# B&R Automation Studio project NAEUL004C00R13L518F00 (part 26)

#### Act_OptP1026Lifter2FBCtrl.st
```iecst
ACTION Act_OptP1026Lifter2FBCtrl:

	fbJogSlowToFastDlyTm.PT	:= T#2s;
	fbJogSlowToFastDlyTm;
	fbLmtRstTm;

	//Lifter Safety Sensor Interruption
	IF EDGENEG(p_tyDI.bLifterSafetyLmtSW1 AND p_tyDI.bLifterSafetyLmtSW2 AND p_tyDI.bLifterTimingBeltSen) THEN
		tyP1026McSetTeach.tyMotionStdLifter.tyBtnStop.bRtCompl	:= TRUE;
	END_IF

	IF EDGEPOS((p_udiLifter2AxisErrID = 21570 OR p_udiLifter2AxisErrID = 21571) AND tyP1026McSetTeach.tyMotionStdLifter.tyBtnJogDown.bValue = FALSE AND tyP1026McSetTeach.tyMotionStdLifter.tyBtnJogUp.bValue = FALSE) THEN
		fbLmtRstTm.IN	:= TRUE;
	END_IF

	IF fbLmtRstTm.Q = TRUE THEN
		tyP1026McSetTeach.tyMotionStdLifter.tyBtnRst.bRtCompl	:= TRUE;
	END_IF

	IF (tyP1026McSetTeach.tyMotionStdLifter.tyBtnJogUp.bValue = FALSE AND tyP1026McSetTeach.tyMotionStdLifter.tyBtnJogDown.bValue = FALSE) AND (p_bLifter2Jogging = TRUE) THEN
		bJogStopLifter	:= TRUE;
	END_IF

	IF tyP1026McSetTeach.tyMotionStdLifter.tyBtnStop.bRtCompl = TRUE THEN
		eLifter2Act		:= LifterActStop;

		IF p_eLifter2Stat = LifterActStop AND p_eLifter2Status = Done THEN
			eLifter2Act	:= LifterActIdle;

			tyP1026McSetTeach.tyMotionStdLifter.tyBtnStop.bRtCompl			:= FALSE;
			tyP1026McSetTeach.tyMotionStdLifter.tyBtnJogDown.bRtCompl		:= FALSE;
			tyP1026McSetTeach.tyMotionStdLifter.tyBtnJogUp.bRtCompl			:= FALSE;
			tyP1026McSetTeach.tyMotionStdLifter.tyBtnOrigin.bRtCompl		:= FALSE;
			tyP1026McSetTeach.tyMotionStdLifter.tyBtnMovAbs.bRtCompl		:= FALSE;
			tyP1026McSetTeach.tyMotionStdLifter.tyBtnMovRel.bRtCompl		:= FALSE;

			tyP1026McSetTeach.tyTeachLifterTopPos2.tyBtn2.bRtCompl				:= FALSE;//
			tyP1026McSetTeach.tyTeachLifterBtmPos2.tyBtn2.bRtCompl				:= FALSE;//

			tyP1026McSetTeach.tyMotionStdLifter.tyBtnStop.bValue			:= TRUE;
			tyP1026McSetTeach.tyMotionStdLifter.tyBtnJogDown.bValue			:= FALSE;
			tyP1026McSetTeach.tyMotionStdLifter.tyBtnJogUp.bValue			:= FALSE;
			tyP1026McSetTeach.tyMotionStdLifter.tyBtnOrigin.bValue			:= FALSE;
			tyP1026McSetTeach.tyMotionStdLifter.tyBtnMovAbs.bValue			:= FALSE;
			tyP1026McSetTeach.tyMotionStdLifter.tyBtnMovRel.bValue			:= FALSE;

			tyP1026McSetTeach.tyTeachLifterTopPos2.tyBtn2.bValue				:= FALSE;
			tyP1026McSetTeach.tyTeachLifterBtmPos2.tyBtn2.bValue				:= FALSE;

			tyP1026McSetTeach.tyMotionStdLifter.tyBtnStop.bRtLk				:= TRUE;
			tyP1026McSetTeach.tyMotionStdLifter.tyBtnJogDown.bRtLk			:= FALSE;
			tyP1026McSetTeach.tyMotionStdLifter.tyBtnJogUp.bRtLk			:= FALSE;
			tyP1026McSetTeach.tyMotionStdLifter.tyBtnOrigin.bRtLk			:= FALSE;
			tyP1026McSetTeach.tyMotionStdLifter.tyBtnMovAbs.bRtLk			:= FALSE;
			tyP1026McSetTeach.tyMotionStdLifter.tyBtnMovRel.bRtLk			:= FALSE;

			tyP1026McSetTeach.tyTeachLifterTopPos2.tyBtn2.bRtLk				:= FALSE;
			tyP1026McSetTeach.tyTeachLifterBtmPos2.tyBtn2.bRtLk				:= FALSE;

		END_IF

	ELSIF (tyP1026McSetTeach.tyMotionStdLifter.tyBtnJogDown.bRtCompl = TRUE) OR (tyP1026McSetTeach.tyMotionStdLifter.tyBtnJogUp.bRtCompl = TRUE) OR (bJogStopLifter = TRUE) THEN
		bJogSlow					:= FALSE;
		bJogFast					:= FALSE;
		fbJogSlowToFastDlyTm.IN		:= FALSE;

		eLifter2Act	:= LifterActJogStop;

		IF p_eLifter2Stat = LifterActJogStop AND p_eLifter2Status = Done THEN
			eLifter2Act		:= LifterActIdle;

			bJogStopLifter	:= FALSE;

			tyP1026McSetTeach.tyMotionStdLifter.tyBtnStop.bRtCompl			:= FALSE;
			tyP1026McSetTeach.tyMotionStdLifter.tyBtnJogDown.bRtCompl		:= FALSE;
			tyP1026McSetTeach.tyMotionStdLifter.tyBtnJogUp.bRtCompl			:= FALSE;
			tyP1026McSetTeach.tyMotionStdLifter.tyBtnOrigin.bRtCompl		:= FALSE;
			tyP1026McSetTeach.tyMotionStdLifter.tyBtnMovAbs.bRtCompl		:= FALSE;
			tyP1026McSetTeach.tyMotionStdLifter.tyBtnMovRel.bRtCompl		:= FALSE;

			tyP1026McSetTeach.tyTeachLifterTopPos2.tyBtn2.bRtCompl				:= FALSE;//
			tyP1026McSetTeach.tyTeachLifterBtmPos2.tyBtn2.bRtCompl				:= FALSE;//

			tyP1026McSetTeach.tyMotionStdLifter.tyBtnStop.bValue			:= TRUE;
			tyP1026McSetTeach.tyMotionStdLifter.tyBtnJogDown.bValue			:= FALSE;
			tyP1026McSetTeach.tyMotionStdLifter.tyBtnJogUp.bValue			:= FALSE;
			tyP1026McSetTeach.tyMotionStdLifter.tyBtnOrigin.bValue			:= FALSE;
			tyP1026McSetTeach.tyMotionStdLifter.tyBtnMovAbs.bValue			:= FALSE;
			tyP1026McSetTeach.tyMotionStdLifter.tyBtnMovRel.bValue			:= FALSE;

			tyP1026McSetTeach.tyTeachLifterTopPos2.tyBtn2.bValue				:= FALSE;
			tyP1026McSetTeach.tyTeachLifterBtmPos2.tyBtn2.bValue				:= FALSE;

			tyP1026McSetTeach.tyMotionStdLifter.tyBtnStop.bRtLk				:= TRUE;
			tyP1026McSetTeach.tyMotionStdLifter.tyBtnJogDown.bRtLk			:= FALSE;
			tyP1026McSetTeach.tyMotionStdLifter.tyBtnJogUp.bRtLk			:= FALSE;
			tyP1026McSetTeach.tyMotionStdLifter.tyBtnOrigin.bRtLk			:= FALSE;
			tyP1026McSetTeach.tyMotionStdLifter.tyBtnMovAbs.bRtLk			:= FALSE;
			tyP1026McSetTeach.tyMotionStdLifter.tyBtnMovRel.bRtLk			:= FALSE;

			tyP1026McSetTeach.tyTeachLifterTopPos2.tyBtn2.bRtLk				:= FALSE;
			tyP1026McSetTeach.tyTeachLifterBtmPos2.tyBtn2.bRtLk				:= FALSE;

		END_IF

	ELSIF tyP1026McSetTeach.tyMotionStdLifter.tyBtnPwr.bRtCompl = TRUE THEN
		tyP1026McSetTeach.tyMotionStdLifter.tyBtnPwr.bRtLk	:= TRUE;

		IF tyP1026McSetTeach.tyMotionStdLifter.tyBtnPwr.bValue = TRUE THEN
			eLifter2Act	:= LifterActPwrOn;

			IF p_eLifter2Stat = LifterActPwrOn AND p_eLifter2Status = Done THEN
				eLifter2Act	:= LifterActIdle;

				tyP1026McSetTeach.tyMotionStdLifter.tyBtnPwr.bRtCompl	:= FALSE;
				tyP1026McSetTeach.tyMotionStdLifter.tyBtnPwr.bRtLk		:= FALSE;
			END_IF
		ELSE
			eLifter2Act	:= LifterActPwrOff;

			IF p_eLifter2Stat = LifterActPwrOff AND p_eLifter2Status = Done THEN
				eLifter2Act	:= LifterActIdle;

				tyP1026McSetTeach.tyMotionStdLifter.tyBtnPwr.bRtCompl	:= FALSE;
				tyP1026McSetTeach.tyMotionStdLifter.tyBtnPwr.bRtLk		:= FALSE;
			END_IF
		END_IF

	ELSIF tyP1026McSetTeach.tyMotionStdLifter.tyBtnOrigin.bRtCompl = TRUE THEN
		tyP1026McSetTeach.tyMotionStdLifter.tyBtnOrigin.bValue	:= TRUE;
		tyP1026McSetTeach.tyMotionStdLifter.tyBtnStop.bValue	:= FALSE;

		tyP1026McSetTeach.tyMotionStdLifter.tyBtnOrigin.bRtLk	:= TRUE;
		tyP1026McSetTeach.tyMotionStdLifter.tyBtnStop.bRtLk		:= FALSE;

		eLifter2Act	:= LifterActHoming;

		IF p_eLifter2Stat = LifterActHoming AND p_eLifter2Status = Done THEN
			eLifter2Act	:= LifterActIdle;

			tyP1026McSetTeach.tyMotionStdLifter.tyBtnOrigin.bRtCompl	:= FALSE;
			tyP1026McSetTeach.tyMotionStdLifter.tyBtnOrigin.bValue		:= FALSE;
			tyP1026McSetTeach.tyMotionStdLifter.tyBtnStop.bValue		:= TRUE;

			tyP1026McSetTeach.tyMotionStdLifter.tyBtnOrigin.bRtLk		:= FALSE;
			tyP1026McSetTeach.tyMotionStdLifter.tyBtnStop.bRtLk			:= TRUE;

		END_IF

	ELSIF tyP1026McSetTeach.tyMotionStdLifter.tyBtnRst.bRtCompl = TRUE THEN
		tyP1026McSetTeach.tyMotionStdLifter.tyBtnRst.bValue	:= TRUE;
		tyP1026McSetTeach.tyMotionStdLifter.tyBtnRst.bRtLk	:= TRUE;

		eLifter2Act	:= LifterActRstAxisErr;

		IF p_eLifter2Stat = LifterActRstAxisErr AND p_eLifter2Status = Done THEN
			eLifter2Act	:= LifterActIdle;

			tyP1026McSetTeach.tyMotionStdLifter.tyBtnRst.bRtCompl	:= FALSE;
			tyP1026McSetTeach.tyMotionStdLifter.tyBtnRst.bValue		:= FALSE;
			tyP1026McSetTeach.tyMotionStdLifter.tyBtnRst.bRtLk		:= FALSE;

			fbLmtRstTm.IN	:= FALSE;
		END_IF

	ELSIF tyP1026McSetTeach.tyTeachLifterTopPos2.tyBtn2.bRtCompl = TRUE THEN
		tyP1026McSetTeach.tyTeachLifterTopPos2.tyBtn2.bValue		:= TRUE;
		tyP1026McSetTeach.tyMotionStdLifter.tyBtnStop.bValue	:= FALSE;

		tyP1026McSetTeach.tyTeachLifterTopPos2.tyBtn2.bRtLk		:= TRUE;
		tyP1026McSetTeach.tyMotionStdLifter.tyBtnStop.bRtLk		:= FALSE;

		diMnlLifterNomSpd2	:= tyP1026McSetTeach.tyMotionStdLifter.tyNumNomSpd.diValue;

		eLifter2Act		:= LifterActGoGPos;

		IF p_eLifter2Stat = LifterActGoGPos AND p_eLifter2Status = Done THEN
			eLifter2Act	:= LifterActIdle;

			tyP1026McSetTeach.tyTeachLifterTopPos2.tyBtn2.bRtCompl		:= FALSE;
			tyP1026McSetTeach.tyTeachLifterTopPos2.tyBtn2.bValue		:= FALSE;
			tyP1026McSetTeach.tyMotionStdLifter.tyBtnStop.bValue	:= TRUE;

			tyP1026McSetTeach.tyTeachLifterTopPos2.tyBtn2.bRtLk		:= FALSE;
			tyP1026McSetTeach.tyMotionStdLifter.tyBtnStop.bRtLk		:= TRUE;
		END_IF

	ELSIF tyP1026McSetTeach.tyTeachLifterBtmPos2.tyBtn2.bRtCompl = TRUE THEN
		tyP1026McSetTeach.tyTeachLifterBtmPos2.tyBtn2.bValue		:= TRUE;
		tyP1026McSetTeach.tyMotionStdLifter.tyBtnStop.bValue	:= FALSE;

		tyP1026McSetTeach.tyTeachLifterBtmPos2.tyBtn2.bRtLk		:= TRUE;
		tyP1026McSetTeach.tyMotionStdLifter.tyBtnStop.bRtLk		:= FALSE;

		diMnlLifterNomSpd2	:= tyP1026McSetTeach.tyMotionStdLifter.tyNumNomSpd.diValue;

		eLifter2Act		:= LifterActGoHPos;

		IF p_eLifter2Stat = LifterActGoHPos AND p_eLifter2Status = Done THEN
			eLifter2Act	:= LifterActIdle;

			tyP1026McSetTeach.tyTeachLifterBtmPos2.tyBtn2.bRtCompl		:= FALSE;
			tyP1026McSetTeach.tyTeachLifterBtmPos2.tyBtn2.bValue		:= FALSE;
			tyP1026McSetTeach.tyMotionStdLifter.tyBtnStop.bValue	:= TRUE;

			tyP1026McSetTeach.tyTeachLifterBtmPos2.tyBtn2.bRtLk		:= FALSE;
			tyP1026McSetTeach.tyMotionStdLifter.tyBtnStop.bRtLk		:= TRUE;
		END_IF

	ELSIF tyP1026McSetTeach.tyMotionStdLifter.tyBtnMovAbs.bRtCompl = TRUE THEN

		tyP1026McSetTeach.tyMotionStdLifter.tyBtnMovAbs.bValue	:= TRUE;
		tyP1026McSetTeach.tyMotionStdLifter.tyBtnStop.bValue	:= FALSE;

		tyP1026McSetTeach.tyMotionStdLifter.tyBtnMovAbs.bRtLk	:= TRUE;
		tyP1026McSetTeach.tyMotionStdLifter.tyBtnStop.bRtLk		:= FALSE;

		diMnlLifterTargetPos2	:= tyP1026McSetTeach.tyMotionStdLifter.tyNumTargetPos.diValue;
		diMnlLifterNomSpd2		:= tyP1026McSetTeach.tyMotionStdLifter.tyNumNomSpd.diValue;

		eLifter2Act			:= LifterActMovAbs;

		IF p_eLifter2Stat = LifterActMovAbs AND p_eLifter2Status = Done THEN
			eLifter2Act	:= LifterActIdle;

			tyP1026McSetTeach.tyMotionStdLifter.tyBtnMovAbs.bRtCompl	:= FALSE;
			tyP1026McSetTeach.tyMotionStdLifter.tyBtnMovAbs.bValue		:= FALSE;
			tyP1026McSetTeach.tyMotionStdLifter.tyBtnStop.bValue		:= TRUE;

			tyP1026McSetTeach.tyMotionStdLifter.tyBtnMovAbs.bRtLk		:= FALSE;
			tyP1026McSetTeach.tyMotionStdLifter.tyBtnStop.bRtLk			:= TRUE;
		END_IF

	ELSIF tyP1026McSetTeach.tyMotionStdLifter.tyBtnMovRel.bRtCompl = TRUE THEN
		tyP1026McSetTeach.tyMotionStdLifter.tyBtnMovRel.bValue			:= TRUE;
		tyP1026McSetTeach.tyMotionStdLifter.tyBtnStop.bValue			:= FALSE;

		tyP1026McSetTeach.tyMotionStdLifter.tyBtnMovRel.bRtLk			:= TRUE;
		tyP1026McSetTeach.tyMotionStdLifter.tyBtnStop.bRtLk				:= FALSE;

		diMnlLifterStepSize2		:= tyP1026McSetTeach.tyMotionStdLifter.tyNumStepSize.diValue;
		diMnlLifterNomSpd2		:= tyP1026McSetTeach.tyMotionStdLifter.tyNumNomSpd.diValue;

		eLifter2Act		:= LifterActMovRel;

		IF p_eLifter2Stat = LifterActMovRel AND p_eLifter2Status = Done THEN
			eLifter2Act	:= LifterActIdle;

			tyP1026McSetTeach.tyMotionStdLifter.tyBtnMovRel.bRtCompl		:= FALSE;
			tyP1026McSetTeach.tyMotionStdLifter.tyBtnMovRel.bValue			:= FALSE;
			tyP1026McSetTeach.tyMotionStdLifter.tyBtnStop.bValue			:= TRUE;

			tyP1026McSetTeach.tyMotionStdLifter.tyBtnMovRel.bRtLk			:= FALSE;
			tyP1026McSetTeach.tyMotionStdLifter.tyBtnStop.bRtLk				:= TRUE;

		END_IF

	ELSIF (tyP1026McSetTeach.tyMotionStdLifter.tyBtnJogDown.bValue = TRUE) AND (fbJogSlowToFastDlyTm.Q = FALSE) AND (bJogSlow = FALSE) THEN
		tyP1026McSetTeach.tyMotionStdLifter.tyBtnStop.bValue				:= FALSE;
		tyP1026McSetTeach.tyMotionStdLifter.tyBtnStop.bRtLk				:= FALSE;

		fbJogSlowToFastDlyTm.IN		:= TRUE;

		diMnlLifterJogSpd2	:= tyP1026McSetTeach.tyMotionStdLifter.tyNumSlwSpd.diValue;

		eLifter2Act		:= LifterActJogDown;

		IF p_eLifter2Stat = LifterActJogDown AND p_eLifter2Status = Done THEN

			eLifter2Act	:= LifterActIdle;
			bJogSlow				:= TRUE;

		ELSIF p_eLifter2Status = Error THEN

			fbJogSlowToFastDlyTm.IN	:= FALSE;
			bJogSlow				:= TRUE;

		END_IF

	ELSIF (tyP1026McSetTeach.tyMotionStdLifter.tyBtnJogDown.bValue = TRUE) AND (fbJogSlowToFastDlyTm.Q = TRUE) AND (bJogFast = FALSE) THEN
		tyP1026McSetTeach.tyMotionStdLifter.tyBtnStop.bValue					:= FALSE;
		tyP1026McSetTeach.tyMotionStdLifter.tyBtnStop.bRtLk					:= FALSE;

		fbJogSlowToFastDlyTm.IN		:= TRUE;

		diMnlLifterJogSpd2	:= tyP1026McSetTeach.tyMotionStdLifter.tyNumNomSpd.diValue;

		eLifter2Act		:= LifterActJogDown;

		IF p_eLifter2Stat = LifterActJogDown AND p_eLifter2Status = Done THEN
			eLifter2Act	:= LifterActIdle;
			bJogFast				:= TRUE;
		ELSIF p_eLifter2Status = Error THEN
			fbJogSlowToFastDlyTm.IN	:= FALSE;
			bJogFast				:= TRUE;
		END_IF

	ELSIF (tyP1026McSetTeach.tyMotionStdLifter.tyBtnJogUp.bValue = TRUE) AND (fbJogSlowToFastDlyTm.Q = FALSE) AND (bJogSlow = FALSE) THEN
		tyP1026McSetTeach.tyMotionStdLifter.tyBtnStop.bValue				:= FALSE;
		tyP1026McSetTeach.tyMotionStdLifter.tyBtnStop.bRtLk				:= FALSE;

		fbJogSlowToFastDlyTm.IN		:= TRUE;

		diMnlLifterJogSpd2	:= tyP1026McSetTeach.tyMotionStdLifter.tyNumSlwSpd.diValue;

		eLifter2Act		:= LifterActJogUp;

		IF p_eLifter2Stat = LifterActJogUp AND p_eLifter2Status = Done THEN
			eLifter2Act	:= LifterActIdle;
			bJogSlow				:= TRUE;

		ELSIF p_eLifter2Status = Error THEN
			fbJogSlowToFastDlyTm.IN	:= FALSE;
			bJogSlow				:= TRUE;
		END_IF

	ELSIF (tyP1026McSetTeach.tyMotionStdLifter.tyBtnJogUp.bValue = TRUE) AND (fbJogSlowToFastDlyTm.Q = TRUE) AND (bJogFast = FALSE) THEN

		tyP1026McSetTeach.tyMotionStdLifter.tyBtnStop.bValue				:= FALSE;
		tyP1026McSetTeach.tyMotionStdLifter.tyBtnStop.bRtLk					:= FALSE;

		fbJogSlowToFastDlyTm.IN		:= TRUE;

		diMnlLifterJogSpd2	:= tyP1026McSetTeach.tyMotionStdLifter.tyNumNomSpd.diValue;

		eLifter2Act		:= LifterActJogUp;

		IF p_eLifter2Stat = LifterActJogUp AND p_eLifter2Status = Done THEN
			eLifter2Act	:= LifterActIdle;
			bJogFast	:= TRUE;

		ELSIF p_eLifter2Status = Error THEN
			fbJogSlowToFastDlyTm.IN	:= FALSE;
			bJogFast				:= TRUE;
		END_IF
	END_IF

	IF tyP1026McSetTeach.tyInOutletShutterFB.tyBtnOpen.bRtCompl = TRUE THEN
		tyP1026McSetTeach.tyInOutletShutterFB.tyBtnOpen.bRtCompl	:= FALSE;

		tyP1026McSetTeach.tyInOutletShutterFB.tyBtnOpen.bValue	:= TRUE;
		tyP1026McSetTeach.tyInOutletShutterFB.tyBtnClose.bValue	:= FALSE;

	ELSIF tyP1026McSetTeach.tyInOutletShutterFB.tyBtnClose.bRtCompl = TRUE THEN
		tyP1026McSetTeach.tyInOutletShutterFB.tyBtnClose.bRtCompl	:= FALSE;

		tyP1026McSetTeach.tyInOutletShutterFB.tyBtnClose.bValue	:= TRUE;
		tyP1026McSetTeach.tyInOutletShutterFB.tyBtnOpen.bValue	:= FALSE;
	END_IF

	IF tyP1026McSetTeach.tyInOutletShutterFB.tyBtnOpen.bValue = TRUE THEN
		eInShutterAct	:= PneuActRet;
		eOutShutterAct	:= PneuActRet;
		eOutShutterAct2	:= PneuActRet;
		eOutShutterAct3	:= PneuActRet;

		IF (p_eInShutterStat = PneuActRet AND p_eInShutterStatus = Done)
			AND (p_eOutShutterStat = PneuActRet AND p_eOutShutterStatus = Done)
			AND (p_eOutShutterStat2 = PneuActRet AND p_eOutShutterStatus2 = Done)
			AND (p_eOutShutterStat3 = PneuActRet AND p_eOutShutterStatus3 = Done)
			THEN
			eInShutterAct	:= PneuActIdle;
			eOutShutterAct	:= PneuActIdle;
			eOutShutterAct2	:= PneuActIdle;
			eOutShutterAct3	:= PneuActIdle;
			tyP1026McSetTeach.tyInOutletShutterFB.tyBtnOpen.bValue	:= FALSE;
		ELSIF p_eInShutterStatus = Error OR p_eOutShutterStatus = Error OR p_eOutShutterStatus2 = Error OR p_eOutShutterStatus3 = Error THEN
			tyP1026McSetTeach.tyInOutletShutterFB.tyBtnOpen.bValue	:= FALSE;
		END_IF

	ELSIF tyP1026McSetTeach.tyInOutletShutterFB.tyBtnClose.bValue = TRUE THEN
		eInShutterAct	:= PneuActExt;
		eOutShutterAct	:= PneuActExt;
		eOutShutterAct2	:= PneuActExt;
		eOutShutterAct3	:= PneuActExt;

		IF (p_eInShutterStat = PneuActExt AND p_eInShutterStatus = Done)
			AND (p_eOutShutterStat = PneuActExt AND p_eOutShutterStatus = Done)
			AND (p_eOutShutterStat2 = PneuActExt AND p_eOutShutterStatus2 = Done)
			AND (p_eOutShutterStat3 = PneuActExt AND p_eOutShutterStatus3 = Done)
			THEN
			eInShutterAct	:= PneuActIdle;
			eOutShutterAct	:= PneuActIdle;
			eOutShutterAct2	:= PneuActIdle;
			eOutShutterAct3	:= PneuActIdle;
			tyP1026McSetTeach.tyInOutletShutterFB.tyBtnClose.bValue := FALSE;
		ELSIF p_eInShutterStatus = Error OR p_eOutShutterStatus = Error OR p_eOutShutterStatus2 = Error OR p_eOutShutterStatus3 = Error THEN
			tyP1026McSetTeach.tyInOutletShutterFB.tyBtnClose.bValue := FALSE;
		END_IF
	END_IF

	IF p_eLifter2Stat = LifterActStop AND (p_eLifter2Status = Done OR p_eLifter2Status = Error) THEN
		eLifter2Act	:= LifterActIdle;
	END_IF

END_ACTION
```

#### Act_OptP1026Lifter2FBStat.st
```iecst
ACTION Act_OptP1026Lifter2FBStat:

	IF p_bLifter2AxisErr = TRUE THEN
		tyP1026McSetTeach.tyMotionStdLifter.tyStringStat.sValue		:= p_sLifter2AxisErrTxt;
	ELSE
		tyP1026McSetTeach.tyMotionStdLifter.tyStringStat.sValue		:= p_sLifter2StatTxt;
	END_IF

END_ACTION
```

#### Act_OptP1026Lifter2Mask.st
```iecst
ACTION Act_OptP1026Lifter2Mask:

	// Interlock Power
	IF p_bLifter2AxisErr = TRUE AND p_bLifter2PwrOn = FALSE THEN
		fUIInRtStatOff(ADR(tyP1026McSetTeach.tyMotionStdLifter.tyBtnPwr.uiMaskRtStat));
		tyP1026McSetTeach.tyMotionStdLifter.tyBtnPwr.bValue		:= FALSE;
	ELSE
		fUIInRtStatHide(ADR(tyP1026McSetTeach.tyMotionStdLifter.tyBtnPwr.uiMaskRtStat));
	END_IF

	// Interlock Others Move
	IF p_bLifter2AxisErr = TRUE OR p_bLifter2PwrOn = FALSE THEN
		fUIInRtStatOff(ADR(tyP1026McSetTeach.tyMotionStdLifter.tyBtnOrigin.uiMaskRtStat));
		fUIInRtStatOff(ADR(tyP1026McSetTeach.tyMotionStdLifter.tyBtnMovRel.uiMaskRtStat));
		fUIInRtStatOff(ADR(tyP1026McSetTeach.tyMotionStdLifter.tyBtnJogUp.uiMaskRtStat));
		fUIInRtStatOff(ADR(tyP1026McSetTeach.tyMotionStdLifter.tyBtnJogDown.uiMaskRtStat));
	ELSE
		fUIInRtStatHide(ADR(tyP1026McSetTeach.tyMotionStdLifter.tyBtnOrigin.uiMaskRtStat));
		fUIInRtStatHide(ADR(tyP1026McSetTeach.tyMotionStdLifter.tyBtnMovRel.uiMaskRtStat));
		fUIInRtStatHide(ADR(tyP1026McSetTeach.tyMotionStdLifter.tyBtnJogUp.uiMaskRtStat));
		fUIInRtStatHide(ADR(tyP1026McSetTeach.tyMotionStdLifter.tyBtnJogDown.uiMaskRtStat));
	END_IF

	// Interlock Move Absolute
	IF p_bLifter2AxisErr = TRUE OR p_bLifter2PwrOn = FALSE OR p_bLifter2IsHomed = FALSE THEN

		fUIInRtStatOff(ADR(tyP1026McSetTeach.tyTeachLifterTopPos2.tyBtn2.uiMaskRtStat));
		fUIInRtStatOff(ADR(tyP1026McSetTeach.tyTeachLifterBtmPos2.tyBtn2.uiMaskRtStat));
		fUIInRtStatOff(ADR(tyP1026McSetTeach.tyMotionStdLifter.tyBtnMovAbs.uiMaskRtStat));
	ELSE
		fUIInRtStatHide(ADR(tyP1026McSetTeach.tyTeachLifterTopPos2.tyBtn2.uiMaskRtStat));
		fUIInRtStatHide(ADR(tyP1026McSetTeach.tyTeachLifterBtmPos2.tyBtn2.uiMaskRtStat));
		fUIInRtStatHide(ADR(tyP1026McSetTeach.tyMotionStdLifter.tyBtnMovAbs.uiMaskRtStat));
	END_IF

	//Interlock Limit Sensor
	IF tyP1026McSetTeach.tyMotionStdLifter.tyBtnDownLmtSen.bValue = TRUE THEN
		fUIInRtStatOff(ADR(tyP1026McSetTeach.tyMotionStdLifter.tyBtnJogDown.uiMaskRtStat));
	END_IF

	IF tyP1026McSetTeach.tyMotionStdLifter.tyBtnUpLmtSen.bValue = TRUE THEN
		fUIInRtStatOff(ADR(tyP1026McSetTeach.tyMotionStdLifter.tyBtnJogUp.uiMaskRtStat));
	END_IF

	// Interlock When Moving
	IF tyP1026McSetTeach.tyMotionStdLifter.tyBtnOrigin.bRtCompl = TRUE THEN
		fUIInRtStatOff(ADR(tyP1026McSetTeach.tyMotionStdLifter.tyBtnMovAbs.uiMaskRtStat));
		fUIInRtStatOff(ADR(tyP1026McSetTeach.tyMotionStdLifter.tyBtnMovRel.uiMaskRtStat));
		fUIInRtStatOff(ADR(tyP1026McSetTeach.tyMotionStdLifter.tyBtnJogUp.uiMaskRtStat));
		fUIInRtStatOff(ADR(tyP1026McSetTeach.tyMotionStdLifter.tyBtnJogDown.uiMaskRtStat));

		fUIInRtStatOff(ADR(tyP1026McSetTeach.tyTeachLifterTopPos2.tyBtn2.uiMaskRtStat));
		fUIInRtStatOff(ADR(tyP1026McSetTeach.tyTeachLifterBtmPos2.tyBtn2.uiMaskRtStat));

	ELSIF tyP1026McSetTeach.tyMotionStdLifter.tyBtnMovAbs.bRtCompl = TRUE THEN
		fUIInRtStatOff(ADR(tyP1026McSetTeach.tyMotionStdLifter.tyBtnOrigin.uiMaskRtStat));
		fUIInRtStatOff(ADR(tyP1026McSetTeach.tyMotionStdLifter.tyBtnMovRel.uiMaskRtStat));
		fUIInRtStatOff(ADR(tyP1026McSetTeach.tyMotionStdLifter.tyBtnJogUp.uiMaskRtStat));
		fUIInRtStatOff(ADR(tyP1026McSetTeach.tyMotionStdLifter.tyBtnJogDown.uiMaskRtStat));

		fUIInRtStatOff(ADR(tyP1026McSetTeach.tyTeachLifterTopPos2.tyBtn2.uiMaskRtStat));
		fUIInRtStatOff(ADR(tyP1026McSetTeach.tyTeachLifterBtmPos2.tyBtn2.uiMaskRtStat));

	ELSIF tyP1026McSetTeach.tyMotionStdLifter.tyBtnMovRel.bRtCompl = TRUE THEN
		fUIInRtStatOff(ADR(tyP1026McSetTeach.tyMotionStdLifter.tyBtnOrigin.uiMaskRtStat));
		fUIInRtStatOff(ADR(tyP1026McSetTeach.tyMotionStdLifter.tyBtnMovAbs.uiMaskRtStat));
		fUIInRtStatOff(ADR(tyP1026McSetTeach.tyMotionStdLifter.tyBtnJogUp.uiMaskRtStat));
		fUIInRtStatOff(ADR(tyP1026McSetTeach.tyMotionStdLifter.tyBtnJogDown.uiMaskRtStat));

		fUIInRtStatOff(ADR(tyP1026McSetTeach.tyTeachLifterTopPos2.tyBtn2.uiMaskRtStat));
		fUIInRtStatOff(ADR(tyP1026McSetTeach.tyTeachLifterBtmPos2.tyBtn2.uiMaskRtStat));

	ELSIF tyP1026McSetTeach.tyMotionStdLifter.tyBtnJogDown.bRtCompl = TRUE OR tyP1026McSetTeach.tyMotionStdLifter.tyBtnJogDown.bValue = TRUE THEN
		fUIInRtStatOff(ADR(tyP1026McSetTeach.tyMotionStdLifter.tyBtnOrigin.uiMaskRtStat));
		fUIInRtStatOff(ADR(tyP1026McSetTeach.tyMotionStdLifter.tyBtnMovAbs.uiMaskRtStat));
		fUIInRtStatOff(ADR(tyP1026McSetTeach.tyMotionStdLifter.tyBtnMovRel.uiMaskRtStat));
		fUIInRtStatOff(ADR(tyP1026McSetTeach.tyMotionStdLifter.tyBtnJogUp.uiMaskRtStat));

		fUIInRtStatOff(ADR(tyP1026McSetTeach.tyTeachLifterTopPos2.tyBtn2.uiMaskRtStat));
		fUIInRtStatOff(ADR(tyP1026McSetTeach.tyTeachLifterBtmPos2.tyBtn2.uiMaskRtStat));

	ELSIF tyP1026McSetTeach.tyMotionStdLifter.tyBtnJogUp.bRtCompl = TRUE OR tyP1026McSetTeach.tyMotionStdLifter.tyBtnJogUp.bValue = TRUE THEN
		fUIInRtStatOff(ADR(tyP1026McSetTeach.tyMotionStdLifter.tyBtnOrigin.uiMaskRtStat));
		fUIInRtStatOff(ADR(tyP1026McSetTeach.tyMotionStdLifter.tyBtnMovAbs.uiMaskRtStat));
		fUIInRtStatOff(ADR(tyP1026McSetTeach.tyMotionStdLifter.tyBtnMovRel.uiMaskRtStat));
		fUIInRtStatOff(ADR(tyP1026McSetTeach.tyMotionStdLifter.tyBtnJogDown.uiMaskRtStat));

		fUIInRtStatOff(ADR(tyP1026McSetTeach.tyTeachLifterTopPos2.tyBtn2.uiMaskRtStat));
		fUIInRtStatOff(ADR(tyP1026McSetTeach.tyTeachLifterBtmPos2.tyBtn2.uiMaskRtStat));

	ELSIF tyP1026McSetTeach.tyTeachLifterTopPos2.tyBtn2.bRtCompl = TRUE THEN
		fUIInRtStatOff(ADR(tyP1026McSetTeach.tyMotionStdLifter.tyBtnOrigin.uiMaskRtStat));
		fUIInRtStatOff(ADR(tyP1026McSetTeach.tyMotionStdLifter.tyBtnMovAbs.uiMaskRtStat));
		fUIInRtStatOff(ADR(tyP1026McSetTeach.tyMotionStdLifter.tyBtnMovRel.uiMaskRtStat));
		fUIInRtStatOff(ADR(tyP1026McSetTeach.tyMotionStdLifter.tyBtnJogUp.uiMaskRtStat));
		fUIInRtStatOff(ADR(tyP1026McSetTeach.tyMotionStdLifter.tyBtnJogDown.uiMaskRtStat));

	ELSIF tyP1026McSetTeach.tyTeachLifterBtmPos2.tyBtn2.bRtCompl = TRUE THEN
		fUIInRtStatOff(ADR(tyP1026McSetTeach.tyMotionStdLifter.tyBtnOrigin.uiMaskRtStat));
		fUIInRtStatOff(ADR(tyP1026McSetTeach.tyMotionStdLifter.tyBtnMovAbs.uiMaskRtStat));
		fUIInRtStatOff(ADR(tyP1026McSetTeach.tyMotionStdLifter.tyBtnMovRel.uiMaskRtStat));
		fUIInRtStatOff(ADR(tyP1026McSetTeach.tyMotionStdLifter.tyBtnJogUp.uiMaskRtStat));
		fUIInRtStatOff(ADR(tyP1026McSetTeach.tyMotionStdLifter.tyBtnJogDown.uiMaskRtStat));

	END_IF

	//Axis Error
	IF tyP1026McSetTeach.tyMotionStdLifter.tyBtnPwr.bRtCompl = TRUE THEN
		fUIInRtStatOff(ADR(tyP1026McSetTeach.tyMotionStdLifter.tyBtnRst.uiMaskRtStat));
	ELSE
		fUIInRtStatHide(ADR(tyP1026McSetTeach.tyMotionStdLifter.tyBtnRst.uiMaskRtStat));
	END_IF

	//Interlock Button Get
	IF p_bLifter2AxisErr = TRUE OR p_bLifter2IsHomed = FALSE OR p_bLifter2FwdLmtSen = TRUE OR p_bLifter2RevLmtSen = TRUE THEN
		fUIInRtStatOff(ADR(tyP1026McSetTeach.tyTeachLifterTopPos2.tyBtn1.uiMaskRtStat));
		fUIInRtStatOff(ADR(tyP1026McSetTeach.tyTeachLifterBtmPos2.tyBtn1.uiMaskRtStat));
	ELSE
		fUIInRtStatHide(ADR(tyP1026McSetTeach.tyTeachLifterTopPos2.tyBtn1.uiMaskRtStat));
		fUIInRtStatHide(ADR(tyP1026McSetTeach.tyTeachLifterBtmPos2.tyBtn1.uiMaskRtStat));
	END_IF

END_ACTION
```

#### Act_OptP1026Lifter2UpdtDat.st
```iecst
ACTION Act_OptP1026Lifter2UpdtDat:

	tyP1026McSetTeach.tyMotionStdLifter.tyNumCurrPos.diValue		:= p_diLifter2ActualPos;
	tyP1026McSetTeach.tyMotionStdLifter.tyNumErrCode.diValue		:= UDINT_TO_DINT(p_udiLifter2AxisErrID);
	tyP1026McSetTeach.tyMotionStdLifter.tyBitmapPwr.usiValueIdx		:= BOOL_TO_USINT(p_bLifter2PwrOn);
	tyP1026McSetTeach.tyMotionStdLifter.tyBitmapRst.usiValueIdx		:= BOOL_TO_USINT(NOT p_bLifter2AxisErr);
	tyP1026McSetTeach.tyMotionStdLifter.tyBitmapOrigin.usiValueIdx	:= BOOL_TO_USINT(p_bLifter2IsHomed);
	tyP1026McSetTeach.tyMotionStdLifter.tyBtnUpLmtSen.bValue		:= p_bLifter2UpSen;
	tyP1026McSetTeach.tyMotionStdLifter.tyBtnDownLmtSen.bValue		:= p_bLifter2DownSen;

	//Machine Bitmap
	IF p_bLifter2IsHomed = TRUE THEN
		IF p_diLifter2ActualPos <= (p_tyNtParamCurr.tyUILifterTargetPos.diMax / 3) THEN
			tyP1026McSetTeach.tyMotionStdLifter.tyBitmapMc.uiValueIdx 	:= 2;
		ELSIF p_diLifter2ActualPos <= (p_tyNtParamCurr.tyUILifterTargetPos.diMax / 3 * 2) THEN
			tyP1026McSetTeach.tyMotionStdLifter.tyBitmapMc.uiValueIdx 	:= 3;
		ELSE
			tyP1026McSetTeach.tyMotionStdLifter.tyBitmapMc.uiValueIdx 	:= 4;
		END_IF
	ELSE
		tyP1026McSetTeach.tyMotionStdLifter.tyBitmapMc.uiValueIdx	:= 2;
	END_IF

	IF p_tyNtParamCurr.eProjMag = ULMagDual THEN
		IF p_tyNtParamCurr.bProjLifterMagPlatform AND p_tyNtParamCurr.bUIConvDirRL THEN
			IF 	tyP1026McSetTeach.tyMotionStdLifter.tyBitmapMc.uiValueIdx < 700 THEN
				tyP1026McSetTeach.tyMotionStdLifter.tyBitmapMc.uiValueIdx	:= tyP1026McSetTeach.tyMotionStdLifter.tyBitmapMc.uiValueIdx + 700;
			END_IF
		ELSIF p_tyNtParamCurr.bProjLifterMagPlatform THEN
			IF p_tyNtParamCurr.bProjMagConvLane2Prep = FALSE THEN
				IF 	tyP1026McSetTeach.tyMotionStdLifter.tyBitmapMc.uiValueIdx < 600 THEN
					tyP1026McSetTeach.tyMotionStdLifter.tyBitmapMc.uiValueIdx	:= tyP1026McSetTeach.tyMotionStdLifter.tyBitmapMc.uiValueIdx + 600;
				END_IF
			ELSE
				IF 	tyP1026McSetTeach.tyMotionStdLifter.tyBitmapMc.uiValueIdx < 903 THEN
					tyP1026McSetTeach.tyMotionStdLifter.tyBitmapMc.uiValueIdx	:= tyP1026McSetTeach.tyMotionStdLifter.tyBitmapMc.uiValueIdx + 903;
				END_IF
			END_IF
		ELSIF p_tyNtParamCurr.bMagAutoVerifyPrep = FALSE THEN
			IF 	tyP1026McSetTeach.tyMotionStdLifter.tyBitmapMc.uiValueIdx < 100 THEN
				tyP1026McSetTeach.tyMotionStdLifter.tyBitmapMc.uiValueIdx	:= tyP1026McSetTeach.tyMotionStdLifter.tyBitmapMc.uiValueIdx + 300;
			END_IF
		ELSE
			IF 	tyP1026McSetTeach.tyMotionStdLifter.tyBitmapMc.uiValueIdx < 300 THEN
				tyP1026McSetTeach.tyMotionStdLifter.tyBitmapMc.uiValueIdx	:= tyP1026McSetTeach.tyMotionStdLifter.tyBitmapMc.uiValueIdx + 300;
			END_IF
		END_IF
	ELSIF p_tyNtParamCurr.eProjMag = ULMagTriple THEN
		IF p_tyNtParamCurr.bProjLifterMagPlatform AND p_tyNtParamCurr.bUIConvDirRL THEN
			IF 	tyP1026McSetTeach.tyMotionStdLifter.tyBitmapMc.uiValueIdx < 800 THEN
				tyP1026McSetTeach.tyMotionStdLifter.tyBitmapMc.uiValueIdx	:= tyP1026McSetTeach.tyMotionStdLifter.tyBitmapMc.uiValueIdx + 800;
			END_IF
		ELSIF p_tyNtParamCurr.bProjLifterMagPlatform THEN
			IF 	tyP1026McSetTeach.tyMotionStdLifter.tyBitmapMc.uiValueIdx < 500 THEN
				tyP1026McSetTeach.tyMotionStdLifter.tyBitmapMc.uiValueIdx	:= tyP1026McSetTeach.tyMotionStdLifter.tyBitmapMc.uiValueIdx + 500;
			END_IF
		ELSIF p_tyNtParamCurr.bMagAutoVerifyPrep = TRUE AND p_tyNtParamCurr.bProjMotorizedPusherPrep = FALSE THEN
			IF 	tyP1026McSetTeach.tyMotionStdLifter.tyBitmapMc.uiValueIdx < 200 THEN
				tyP1026McSetTeach.tyMotionStdLifter.tyBitmapMc.uiValueIdx	:= tyP1026McSetTeach.tyMotionStdLifter.tyBitmapMc.uiValueIdx + 200;
			END_IF
		ELSIF p_tyNtParamCurr.bMagAutoVerifyPrep = FALSE AND p_tyNtParamCurr.bProjMotorizedPusherPrep = TRUE THEN
			IF 	tyP1026McSetTeach.tyMotionStdLifter.tyBitmapMc.uiValueIdx < 400 THEN
				tyP1026McSetTeach.tyMotionStdLifter.tyBitmapMc.uiValueIdx	:= tyP1026McSetTeach.tyMotionStdLifter.tyBitmapMc.uiValueIdx + 400;
			END_IF
		END_IF
	END_IF

END_ACTION
```

#### Act_OptP1026LifterKeypad.st
```iecst
ACTION Act_OptP1026LifterKeypad:

	IF fUIOutRtStatTPIsOpen(ADR(tyP1026McSetTeach.tyMotionStdLifter.tyNumTargetPos.uiRtStat)) = TRUE THEN
		tyProperty.tyKeypad.tyStringTitle.sKeypadTitle		:= tyP1026McSetTeach.tyMotionStdLifter.tyNumTargetPos.sKeypadTitle;

	ELSIF fUIOutRtStatTPIsOpen(ADR(tyP1026McSetTeach.tyMotionStdLifter.tyNumStepSize.uiRtStat)) = TRUE THEN
		tyProperty.tyKeypad.tyStringTitle.sKeypadTitle		:= tyP1026McSetTeach.tyMotionStdLifter.tyNumStepSize.sKeypadTitle;

	ELSIF fUIOutRtStatTPIsOpen(ADR(tyP1026McSetTeach.tyMotionStdLifter.tyNumNomSpd.uiRtStat)) = TRUE THEN
		tyProperty.tyKeypad.tyStringTitle.sKeypadTitle		:= tyP1026McSetTeach.tyMotionStdLifter.tyNumNomSpd.sKeypadTitle;

	ELSIF fUIOutRtStatTPIsOpen(ADR(tyP1026McSetTeach.tyMotionStdLifter.tyNumSlwSpd.uiRtStat)) = TRUE THEN
		tyProperty.tyKeypad.tyStringTitle.sKeypadTitle		:= tyP1026McSetTeach.tyMotionStdLifter.tyNumSlwSpd.sKeypadTitle;

	END_IF

END_ACTION
```

#### Act_OptP1026LifterRstMnl.st
```iecst
ACTION Act_OptP1026LifterRstMnl:

	IF EDGEPOS((bManualMod = FALSE) OR (p_eLifterBtmStatus = Error)) THEN

		bJogSlow				:= FALSE;
		bJogFast				:= FALSE;
		fbJogSlowToFastDlyTm.IN	:= FALSE;

		tyP1026McSetTeach.tyMotionStdLifter.tyBtnPwr.bRtCompl			:= FALSE;
		tyP1026McSetTeach.tyMotionStdLifter.tyBtnStop.bRtCompl			:= FALSE;
		tyP1026McSetTeach.tyMotionStdLifter.tyBtnOrigin.bRtCompl		:= FALSE;
		tyP1026McSetTeach.tyMotionStdLifter.tyBtnRst.bRtCompl			:= FALSE;
		tyP1026McSetTeach.tyMotionStdLifter.tyBtnMovAbs.bRtCompl		:= FALSE;
		tyP1026McSetTeach.tyMotionStdLifter.tyBtnMovRel.bRtCompl		:= FALSE;
		tyP1026McSetTeach.tyMotionStdLifter.tyBtnJogUp.bRtCompl			:= FALSE;
		tyP1026McSetTeach.tyMotionStdLifter.tyBtnJogDown.bRtCompl		:= FALSE;

		tyP1026McSetTeach.tyTeachLifterPosA.tyBtn2.bRtCompl				:= FALSE;
		tyP1026McSetTeach.tyTeachLifterPosB.tyBtn2.bRtCompl				:= FALSE;
		tyP1026McSetTeach.tyTeachLifterTopPos.tyBtn2.bRtCompl				:= FALSE;
		tyP1026McSetTeach.tyTeachLifterBtmPos.tyBtn2.bRtCompl				:= FALSE;
		tyP1026McSetTeach.tyTeachLifterTopPos2.tyBtn2.bRtCompl				:= FALSE;
		tyP1026McSetTeach.tyTeachLifterBtmPos2.tyBtn2.bRtCompl				:= FALSE;

		tyP1026McSetTeach.tyMotionStdLifter.tyBtnPwr.bValue				:= FALSE;
		tyP1026McSetTeach.tyMotionStdLifter.tyBtnStop.bValue			:= TRUE;
		tyP1026McSetTeach.tyMotionStdLifter.tyBtnOrigin.bValue			:= FALSE;
		tyP1026McSetTeach.tyMotionStdLifter.tyBtnRst.bValue				:= FALSE;
		tyP1026McSetTeach.tyMotionStdLifter.tyBtnMovAbs.bValue			:= FALSE;
		tyP1026McSetTeach.tyMotionStdLifter.tyBtnMovRel.bValue			:= FALSE;
		tyP1026McSetTeach.tyMotionStdLifter.tyBtnJogUp.bValue			:= FALSE;
		tyP1026McSetTeach.tyMotionStdLifter.tyBtnJogDown.bValue			:= FALSE;

		tyP1026McSetTeach.tyTeachLifterPosA.tyBtn2.bValue				:= FALSE;
		tyP1026McSetTeach.tyTeachLifterPosB.tyBtn2.bValue				:= FALSE;
		tyP1026McSetTeach.tyTeachLifterTopPos.tyBtn2.bValue				:= FALSE;
		tyP1026McSetTeach.tyTeachLifterBtmPos.tyBtn2.bValue				:= FALSE;
		tyP1026McSetTeach.tyTeachLifterTopPos2.tyBtn2.bValue				:= FALSE;
		tyP1026McSetTeach.tyTeachLifterBtmPos2.tyBtn2.bValue				:= FALSE;

		tyP1026McSetTeach.tyMotionStdLifter.tyBtnPwr.bRtLk				:= FALSE;
		tyP1026McSetTeach.tyMotionStdLifter.tyBtnStop.bRtLk				:= TRUE;
		tyP1026McSetTeach.tyMotionStdLifter.tyBtnOrigin.bRtLk			:= FALSE;
		tyP1026McSetTeach.tyMotionStdLifter.tyBtnRst.bRtLk				:= FALSE;
		tyP1026McSetTeach.tyMotionStdLifter.tyBtnMovAbs.bRtLk			:= FALSE;
		tyP1026McSetTeach.tyMotionStdLifter.tyBtnMovRel.bRtLk			:= FALSE;
		tyP1026McSetTeach.tyMotionStdLifter.tyBtnJogUp.bRtLk			:= FALSE;
		tyP1026McSetTeach.tyMotionStdLifter.tyBtnJogDown.bRtLk			:= FALSE;

		tyP1026McSetTeach.tyTeachLifterPosA.tyBtn2.bRtLk				:= FALSE;
		tyP1026McSetTeach.tyTeachLifterPosB.tyBtn2.bRtLk				:= FALSE;
		tyP1026McSetTeach.tyTeachLifterTopPos.tyBtn2.bRtLk				:= FALSE;
		tyP1026McSetTeach.tyTeachLifterBtmPos.tyBtn2.bRtLk				:= FALSE;
		tyP1026McSetTeach.tyTeachLifterTopPos2.tyBtn2.bRtLk				:= FALSE;
		tyP1026McSetTeach.tyTeachLifterBtmPos2.tyBtn2.bRtLk				:= FALSE;

		tyP1026McSetTeach.tyMotionStdLifter.tyBtnPwr.uiMaskRtStat		:= TRUE;
		tyP1026McSetTeach.tyMotionStdLifter.tyBtnOrigin.uiMaskRtStat	:= FALSE;
		tyP1026McSetTeach.tyMotionStdLifter.tyBtnRst.uiMaskRtStat		:= TRUE;
		tyP1026McSetTeach.tyMotionStdLifter.tyBtnMovAbs.uiMaskRtStat	:= FALSE;
		tyP1026McSetTeach.tyMotionStdLifter.tyBtnMovRel.uiMaskRtStat	:= FALSE;
		tyP1026McSetTeach.tyMotionStdLifter.tyBtnJogUp.uiMaskRtStat		:= FALSE;
		tyP1026McSetTeach.tyMotionStdLifter.tyBtnJogDown.uiMaskRtStat	:= FALSE;

		tyP1026McSetTeach.tyTeachLifterPosA.tyBtn2.uiMaskRtStat			:= FALSE;
		tyP1026McSetTeach.tyTeachLifterPosB.tyBtn2.uiMaskRtStat			:= FALSE;
		tyP1026McSetTeach.tyTeachLifterTopPos.tyBtn2.uiMaskRtStat			:= FALSE;
		tyP1026McSetTeach.tyTeachLifterBtmPos.tyBtn2.uiMaskRtStat			:= FALSE;
		tyP1026McSetTeach.tyTeachLifterTopPos2.tyBtn2.uiMaskRtStat			:= FALSE;
		tyP1026McSetTeach.tyTeachLifterBtmPos2.tyBtn2.uiMaskRtStat			:= FALSE;

		eInShutterAct	:= PneuActIdle;
		eOutShutterAct	:= PneuActIdle;
		eOutShutterAct2	:= PneuActIdle;
		eOutShutterAct3	:= PneuActIdle;

		tyP1026McSetTeach.tyInOutletShutterFB.tyBtnClose.bRtCompl	:= FALSE;
		tyP1026McSetTeach.tyInOutletShutterFB.tyBtnClose.bValue	:= FALSE;
		tyP1026McSetTeach.tyInOutletShutterFB.tyBtnOpen.bRtCompl	:= FALSE;
		tyP1026McSetTeach.tyInOutletShutterFB.tyBtnOpen.bValue	:= FALSE;

	END_IF

END_ACTION
```

#### Act_EntP1030Disp.st
```iecst
ACTION Act_EntP1030Disp:

	//Access Address
	p_tyC0005Main ACCESS ADR(tyCommon.tyMain);

	p_tyC0007Notif ACCESS ADR(tyCommon.tyNotif);

	p_tyC0008MsgBox ACCESS ADR(tyP1030MagSet.tyMsgBoxHide);

	p_tyC0009Info ACCESS ADR(tyCommon.tyInfo);

	p_tyP1030MagSet ACCESS ADR(tyP1030MagSet.tyMagSet);

	IF bTeachTravPosMag1 OR bTeachTravPosMag2 OR bTeachTravPosMag3 OR bTeachLifterMag1Slt1Pos OR bTeachLifterMag2Slt1Pos OR bTeachLifterMag3Slt1Pos THEN
		bTeachTravPosMag1		:= FALSE;
		bTeachTravPosMag2		:= FALSE;
		bTeachTravPosMag3		:= FALSE;
		bTeachLifterMag1Slt1Pos	:= FALSE;
		bTeachLifterMag2Slt1Pos	:= FALSE;
		bTeachLifterMag3Slt1Pos	:= FALSE;
	ELSE
		udiP1030SelectedRowOld	 := 0;
	END_IF

	// Enabling Auto Detect Magazine Model Setting
	tyP1030MagSet.tyMagSet.tyDrpDnMagModel.uiRtStat := NOT(p_tyNtParamCurr.bMagAutoVerifyPrep (*OR p_tyNtParamCurr.bMagSelPrep*));
	tyP1030MagSet.tyMagSet.tyTxtMagModel.uiRtStat	:= NOT(p_tyNtParamCurr.bMagAutoVerifyPrep (*OR p_tyNtParamCurr.bMagSelPrep*));

//	IF p_tyNtParamCurr.bMagAutoVerifyPrep AND NOT p_tyNtParamCurr.bMagSelPrep THEN
		tyP1030MagSet.tyMagSet.tyDrpDnMagModel.usiValueMinIdx	:= 0;
		tyP1030MagSet.tyMagSet.tyDrpDnMagModel.usiValueMaxIdx	:= 2;
		tyP1030MagSet.tyMagSet.tyDrpDnMagModel.usiValueIdx		:= 0;
//	ELSIF NOT p_tyNtParamCurr.bMagAutoVerifyPrep AND p_tyNtParamCurr.bMagSelPrep THEN
//		tyP1030MagSet.tyMagSet.tyDrpDnMagModel.usiValueMinIdx	:= 3;
//		tyP1030MagSet.tyMagSet.tyDrpDnMagModel.usiValueMaxIdx	:= 4;
//		tyP1030MagSet.tyMagSet.tyDrpDnMagModel.usiValueIdx		:= 3;
//	END_IF
	tyP1030MagSet.tyMagSet.tyBtnSort.bValue		:= FALSE;
	tyP1030MagSet.tyMagSet.tyBtnSort.bRtCompl	:= FALSE;
END_ACTION
```

#### Act_OptP1030Mask.st
```iecst
ACTION Act_OptP1030Mask:

	IF tyP1030MagSet.tyMagSet.tyStringRecipeNm.bRtCompl				OR tyP1030MagSet.tyMagSet.tyNumSltToSltDist.bRtCompl
		OR tyP1030MagSet.tyMagSet.tyNumMaxSlt.bRtCompl				OR tyP1030MagSet.tyMagSet.tyNumLifterMag1Slt1Pos.bRtCompl
		OR tyP1030MagSet.tyMagSet.tyNumLifterMag2Slt1Pos.bRtCompl	OR tyP1030MagSet.tyMagSet.tyNumLifterMag3Slt1Pos.bRtCompl
		OR tyP1030MagSet.tyMagSet.tyNumTravPosMag1.bRtCompl			OR tyP1030MagSet.tyMagSet.tyNumTravPosMag2.bRtCompl
		OR tyP1030MagSet.tyMagSet.tyNumTravPosMag3.bRtCompl			OR tyP1030MagSet.tyMagSet.tyDrpDnMagModel.bRtCompl
		OR tyP1030MagSet.tyMagSet.tyNumMagMaxBrdWidth.bRtCompl
		OR tyP1030MagSet.tyMagSet.tyBtnSafetyBarDisabled.bRtCompl
		OR tyP1030MagSet.tyMagSet.tyBtnMagHeightChkEn.bRtCompl
		THEN

		fUIInRtStatHide(ADR(tyP1030MagSet.tyMagSet.tyBtnSave.uiMaskRtStat));

		tyP1030MagSet.tyMagSet.tyStringRecipeNm.bRtCompl		:= FALSE;
		tyP1030MagSet.tyMagSet.tyNumSltToSltDist.bRtCompl		:= FALSE;
		tyP1030MagSet.tyMagSet.tyNumMaxSlt.bRtCompl				:= FALSE;
		tyP1030MagSet.tyMagSet.tyNumLifterMag1Slt1Pos.bRtCompl	:= FALSE;
		tyP1030MagSet.tyMagSet.tyNumLifterMag2Slt1Pos.bRtCompl	:= FALSE;
		tyP1030MagSet.tyMagSet.tyNumLifterMag3Slt1Pos.bRtCompl	:= FALSE;
		tyP1030MagSet.tyMagSet.tyNumTravPosMag1.bRtCompl		:= FALSE;
		tyP1030MagSet.tyMagSet.tyNumTravPosMag2.bRtCompl		:= FALSE;
		tyP1030MagSet.tyMagSet.tyNumTravPosMag3.bRtCompl		:= FALSE;
		tyP1030MagSet.tyMagSet.tyDrpDnMagModel.bRtCompl			:= FALSE;
		tyP1030MagSet.tyMagSet.tyNumMagMaxBrdWidth.bRtCompl		:= FALSE;
		tyP1030MagSet.tyMagSet.tyBtnSafetyBarDisabled.bRtCompl  := FALSE;
		tyP1030MagSet.tyMagSet.tyBtnMagHeightChkEn.bRtCompl		:= FALSE;
	END_IF

	IF tyP1030MagSet.tyMagSet.tyTableRecipe.a_tyStringDataCol1[tyP1030Table.uiSelectedRow].sValue <> '' THEN
		fUIInRtStatHide(ADR(tyP1030MagSet.tyMagSet.tyBtnDelete.uiMaskRtStat));
	ELSE
		fUIInRtStatOff(ADR(tyP1030MagSet.tyMagSet.tyBtnDelete.uiMaskRtStat));
	END_IF

	tyP1030MagSet.tyMagSet.tyBtnSort.uiMaskRtStat.0		:= (tyP1030MagSet.tyMagSet.tyTableRecipe.a_tyStringDataCol1[1].sValue <> '')
	AND (tyP1030MagSet.tyMagSet.tyBtnSave.uiMaskRtStat.0 = FALSE) AND (tyP1030MagSet.tyMagSet.tyBtnDelete.bRtCompl = FALSE) ;

END_ACTION
```

#### Act_OptP1030Save.st
```iecst
ACTION Act_OptP1030Save:

	IF tyP1030MagSet.tyMagSet.tyBtnSave.bRtCompl = TRUE THEN
		IF usiSaveMagRcpStep = 0 THEN
			//Mask Table
			tyP1030MagSet.tyMagSet.tyTableRecipe.uiMaskRtStat				:= FALSE;
			tyP1030MagSet.tyMagSet.tyBtnDelete.uiMaskRtStat					:= FALSE;

			p_tyC0008MsgBox ACCESS ADR(tyP1030MagSet.tyMsgBoxSaveAsk);

			IF tyP1030MagSet.tyMsgBoxSaveAsk.tyBtnYes.bRtCompl = TRUE THEN
				tyP1030MagSet.tyMsgBoxSaveAsk.tyBtnYes.bRtCompl				:= FALSE;
				tyP1030MagSet.tyMsgBoxSaveAsk.tyBtnYes.bValue				:= FALSE;

				p_tyC0008MsgBox ACCESS ADR(tyP1030MagSet.tyMsgBoxHide);

				usiSaveMagRcpStep	:= 1;

			ELSIF tyP1030MagSet.tyMsgBoxSaveAsk.tyBtnNo.bRtCompl = TRUE THEN
				tyP1030MagSet.tyMsgBoxSaveAsk.tyBtnNo.bRtCompl				:= FALSE;
				tyP1030MagSet.tyMsgBoxSaveAsk.tyBtnNo.bValue				:= FALSE;

				p_tyC0008MsgBox ACCESS ADR(tyP1030MagSet.tyMsgBoxHide);

				usiSaveMagRcpStep	:= 99;

			END_IF

		ELSIF usiSaveMagRcpStep = 1 THEN
			tyMagRcpInfoIn.sRcpNm					:= tyP1030MagSet.tyMagSet.tyStringRecipeNm.sValue;
			tyMagRcpInfoIn.diSltToSltInUM			:= tyP1030MagSet.tyMagSet.tyNumSltToSltDist.diValue;
			tyMagRcpInfoIn.diTtlSlt					:= tyP1030MagSet.tyMagSet.tyNumMaxSlt.diValue;
			tyMagRcpInfoIn.diMag1Slt1PosInUM		:= tyP1030MagSet.tyMagSet.tyNumLifterMag1Slt1Pos.diValue;
			tyMagRcpInfoIn.diMag2Slt1PosInUM		:= tyP1030MagSet.tyMagSet.tyNumLifterMag2Slt1Pos.diValue;
			tyMagRcpInfoIn.diMag3Slt1PosInUM		:= tyP1030MagSet.tyMagSet.tyNumLifterMag3Slt1Pos.diValue;
			tyMagRcpInfoIn.diMag1TravPosInUM		:= tyP1030MagSet.tyMagSet.tyNumTravPosMag1.diValue;
			tyMagRcpInfoIn.diMag2TravPosInUM		:= tyP1030MagSet.tyMagSet.tyNumTravPosMag2.diValue;
			tyMagRcpInfoIn.diMag3TravPosInUM		:= tyP1030MagSet.tyMagSet.tyNumTravPosMag3.diValue;
			tyMagRcpInfoIn.usiMagModel				:= tyP1030MagSet.tyMagSet.tyDrpDnMagModel.usiValueIdx;
			tyMagRcpInfoIn.diMagMaxBrdWidth			:= tyP1030MagSet.tyMagSet.tyNumMagMaxBrdWidth.diValue;
			tyMagRcpInfoIn.bSafetyBarDisabled		:= tyP1030MagSet.tyMagSet.tyBtnSafetyBarDisabled.bValue;
			tyMagRcpInfoIn.bMagHeightChkEn			:= tyP1030MagSet.tyMagSet.tyBtnMagHeightChkEn.bValue;

			eMagRcpAct					:= MagRcpActAddEdit;

			IF p_eMagRcpStat = MagRcpActAddEdit AND p_eMagRcpStatus = Done THEN
				eMagRcpAct	:= MagRcpActIdle;

				IF p_bMagRcpNmEmpty = TRUE THEN
					usiSaveMagRcpStep		:= 2;
				ELSIF p_bMagRcpListFull = TRUE THEN
					usiSaveMagRcpStep		:= 3;
				ELSE
					tyP1030MagSet.tyMagSet.tyBtnSort.bValue	:= FALSE;
					bRefreshMagRcpTable	:= TRUE;
					bRefreshMagRcpDetail	:= TRUE;
					usiSaveMagRcpStep		:= 4;
				END_IF

			ELSIF p_eMagRcpStatus = Error THEN
				p_tyC0008MsgBox ACCESS ADR(tyP1030MagSet.tyMsgBoxSaveErr);

				IF tyP1030MagSet.tyMsgBoxSaveErr.tyBtnNo.bRtCompl = TRUE THEN
					tyP1030MagSet.tyMsgBoxSaveErr.tyBtnNo.bRtCompl 		:= FALSE;
					tyP1030MagSet.tyMsgBoxSaveErr.tyBtnNo.bValue 		:= FALSE;

					p_tyC0008MsgBox ACCESS ADR(tyP1030MagSet.tyMsgBoxHide);

					usiSaveMagRcpStep		:= 99;
				END_IF
			END_IF

		// Magazine Recipe Param Error
		ELSIF usiSaveMagRcpStep = 2 THEN
			p_tyC0008MsgBox ACCESS ADR(tyP1030MagSet.tyMsgBoxSaveNoNm);

			IF tyP1030MagSet.tyMsgBoxSaveNoNm.tyBtnNo.bRtCompl = TRUE THEN
				tyP1030MagSet.tyMsgBoxSaveNoNm.tyBtnNo.bRtCompl 			:= FALSE;
				tyP1030MagSet.tyMsgBoxSaveNoNm.tyBtnNo.bValue 				:= FALSE;

				p_tyC0008MsgBox ACCESS ADR(tyP1030MagSet.tyMsgBoxHide);

				usiSaveMagRcpStep		:= 99;
			END_IF

		// Magazine Recipe List Full
		ELSIF usiSaveMagRcpStep = 3 THEN
			p_tyC0008MsgBox ACCESS ADR(tyP1030MagSet.tyMsgBoxListFull);

			IF tyP1030MagSet.tyMsgBoxListFull.tyBtnNo.bRtCompl = TRUE THEN
				tyP1030MagSet.tyMsgBoxListFull.tyBtnNo.bRtCompl 				:= FALSE;
				tyP1030MagSet.tyMsgBoxListFull.tyBtnNo.bValue 					:= FALSE;

				p_tyC0008MsgBox ACCESS ADR(tyP1030MagSet.tyMsgBoxHide);

				usiSaveMagRcpStep		:= 99;
			END_IF

		ELSIF usiSaveMagRcpStep = 4 THEN
			IF tyMagRcpInfoIn.sRcpNm = p_tyMagRcpCurrRcp.sRcpNm THEN
				p_tyC0008MsgBox ACCESS ADR(tyP1030MagSet.tyMsgBoxReloadCurrRcp);

				IF tyP1030MagSet.tyMsgBoxReloadCurrRcp.tyBtnNo.bRtCompl = TRUE THEN
					tyP1030MagSet.tyMsgBoxReloadCurrRcp.tyBtnNo.bRtCompl 	:= FALSE;
					tyP1030MagSet.tyMsgBoxReloadCurrRcp.tyBtnNo.bValue 		:= FALSE;

					p_tyC0008MsgBox ACCESS ADR(tyP1030MagSet.tyMsgBoxHide);

					usiSaveMagRcpStep		:= 99;
				END_IF
			ELSE
				usiSaveMagRcpStep			:= 99;
			END_IF

		ELSIF usiSaveMagRcpStep = 99 THEN
			bRefreshMagRcpTable 			:= FALSE;

			//Unmask
			tyP1030MagSet.tyMagSet.tyTableRecipe.uiMaskRtStat	:= TRUE;
			tyP1030MagSet.tyMagSet.tyBtnDelete.uiMaskRtStat		:= TRUE;

			//Reset
			tyP1030MagSet.tyMagSet.tyBtnSave.bRtCompl	:= FALSE;
			tyP1030MagSet.tyMagSet.tyBtnSave.bValue		:= FALSE;

			usiSaveMagRcpStep	:= 0;

		END_IF

	END_IF

END_ACTION
```

#### Act_OptP1030LoadData.st
```iecst
ACTION Act_OptP1030LoadData:

	udiP1030SelectedRow		:= STRING_TO_UDINT(tyP1030MagSet.tyMagSet.tyTableRecipe.a_tyStringDataCol0[tyP1030Table.uiSelectedRow].sValue);

	IF udiP1030SelectedRow <> udiP1030SelectedRowOld OR bRefreshMagRcpDetail = TRUE OR bUpdateP1030LoadData THEN

		IF tyP1030MagSet.tyMagSet.tyTableRecipe.a_tyStringDataCol1[tyP1030Table.uiSelectedRow].sValue <> '' THEN
			//Update Recipe Data
			IF tyP1030MagSet.tyMagSet.tyBtnSort.bValue THEN
				tyP1030MagSet.tyMagSet.tyStringRecipeNm.sValue			:= p_tyMagRcpSortedList[udiP1030SelectedRow].sRcpNm;
				tyP1030MagSet.tyMagSet.tyNumSltToSltDist.diValue		:= p_tyMagRcpSortedList[udiP1030SelectedRow].diSltToSltInUM;
				tyP1030MagSet.tyMagSet.tyNumMaxSlt.diValue				:= p_tyMagRcpSortedList[udiP1030SelectedRow].diTtlSlt;
				tyP1030MagSet.tyMagSet.tyNumLifterMag1Slt1Pos.diValue	:= p_tyMagRcpSortedList[udiP1030SelectedRow].diMag1Slt1PosInUM;
				tyP1030MagSet.tyMagSet.tyNumLifterMag2Slt1Pos.diValue	:= p_tyMagRcpSortedList[udiP1030SelectedRow].diMag2Slt1PosInUM;
				tyP1030MagSet.tyMagSet.tyNumLifterMag3Slt1Pos.diValue	:= p_tyMagRcpSortedList[udiP1030SelectedRow].diMag3Slt1PosInUM;
				tyP1030MagSet.tyMagSet.tyNumTravPosMag1.diValue			:= p_tyMagRcpSortedList[udiP1030SelectedRow].diMag1TravPosInUM;
				tyP1030MagSet.tyMagSet.tyNumTravPosMag2.diValue			:= p_tyMagRcpSortedList[udiP1030SelectedRow].diMag2TravPosInUM;
				tyP1030MagSet.tyMagSet.tyNumTravPosMag3.diValue			:= p_tyMagRcpSortedList[udiP1030SelectedRow].diMag3TravPosInUM;
				tyP1030MagSet.tyMagSet.tyDrpDnMagModel.usiValueIdx		:= p_tyMagRcpSortedList[udiP1030SelectedRow].usiMagModel;
				tyP1030MagSet.tyMagSet.tyNumMagMaxBrdWidth.diValue		:= p_tyMagRcpSortedList[udiP1030SelectedRow].diMagMaxBrdWidth;
				tyP1030MagSet.tyMagSet.tyBtnSafetyBarDisabled.bValue	:= p_tyMagRcpSortedList[udiP1030SelectedRow].bSafetyBarDisabled;
				tyP1030MagSet.tyMagSet.tyBtnMagHeightChkEn.bValue		:= p_tyMagRcpSortedList[udiP1030SelectedRow].bMagHeightChkEn;
			ELSE
				tyP1030MagSet.tyMagSet.tyStringRecipeNm.sValue			:= p_tyMagRcpCurrList[udiP1030SelectedRow].sRcpNm;
				tyP1030MagSet.tyMagSet.tyNumSltToSltDist.diValue		:= p_tyMagRcpCurrList[udiP1030SelectedRow].diSltToSltInUM;
				tyP1030MagSet.tyMagSet.tyNumMaxSlt.diValue				:= p_tyMagRcpCurrList[udiP1030SelectedRow].diTtlSlt;
				tyP1030MagSet.tyMagSet.tyNumLifterMag1Slt1Pos.diValue	:= p_tyMagRcpCurrList[udiP1030SelectedRow].diMag1Slt1PosInUM;
				tyP1030MagSet.tyMagSet.tyNumLifterMag2Slt1Pos.diValue	:= p_tyMagRcpCurrList[udiP1030SelectedRow].diMag2Slt1PosInUM;
				tyP1030MagSet.tyMagSet.tyNumLifterMag3Slt1Pos.diValue	:= p_tyMagRcpCurrList[udiP1030SelectedRow].diMag3Slt1PosInUM;
				tyP1030MagSet.tyMagSet.tyNumTravPosMag1.diValue			:= p_tyMagRcpCurrList[udiP1030SelectedRow].diMag1TravPosInUM;
				tyP1030MagSet.tyMagSet.tyNumTravPosMag2.diValue			:= p_tyMagRcpCurrList[udiP1030SelectedRow].diMag2TravPosInUM;
				tyP1030MagSet.tyMagSet.tyNumTravPosMag3.diValue			:= p_tyMagRcpCurrList[udiP1030SelectedRow].diMag3TravPosInUM;
				tyP1030MagSet.tyMagSet.tyDrpDnMagModel.usiValueIdx		:= p_tyMagRcpCurrList[udiP1030SelectedRow].usiMagModel;
				tyP1030MagSet.tyMagSet.tyNumMagMaxBrdWidth.diValue		:= p_tyMagRcpCurrList[udiP1030SelectedRow].diMagMaxBrdWidth;
				tyP1030MagSet.tyMagSet.tyBtnSafetyBarDisabled.bValue	:= p_tyMagRcpCurrList[udiP1030SelectedRow].bSafetyBarDisabled;
				tyP1030MagSet.tyMagSet.tyBtnMagHeightChkEn.bValue		:= p_tyMagRcpCurrList[udiP1030SelectedRow].bMagHeightChkEn;
			END_IF
		ELSE

			tyP1030MagSet.tyMagSet.tyStringRecipeNm.sValue			:= '';
			tyP1030MagSet.tyMagSet.tyNumSltToSltDist.diValue		:= 10000;
			tyP1030MagSet.tyMagSet.tyNumMaxSlt.diValue				:= p_tyNtParamCurr.diProjMagMaxSlt;
			tyP1030MagSet.tyMagSet.tyNumLifterMag1Slt1Pos.diValue	:= 0;
			tyP1030MagSet.tyMagSet.tyNumLifterMag2Slt1Pos.diValue	:= 0;
			tyP1030MagSet.tyMagSet.tyNumLifterMag3Slt1Pos.diValue	:= 0;
			tyP1030MagSet.tyMagSet.tyNumTravPosMag1.diValue			:= 0;
			tyP1030MagSet.tyMagSet.tyNumTravPosMag2.diValue			:= 0;
			tyP1030MagSet.tyMagSet.tyNumTravPosMag3.diValue			:= 0;
			tyP1030MagSet.tyMagSet.tyDrpDnMagModel.usiValueIdx		:= 0;
			tyP1030MagSet.tyMagSet.tyNumMagMaxBrdWidth.diValue		:= 0;
			tyP1030MagSet.tyMagSet.tyBtnSafetyBarDisabled.bValue	:= FALSE;
			tyP1030MagSet.tyMagSet.tyBtnMagHeightChkEn.bValue		:= FALSE;
		END_IF

		bRefreshMagRcpDetail	:= FALSE;
		bUpdateP1030LoadData	:= FALSE;
		udiP1030SelectedRowOld 	:= udiP1030SelectedRow;

		fUIInRtStatOff(ADR(tyP1030MagSet.tyMagSet.tyBtnSave.uiMaskRtStat));

	END_IF

END_ACTION
```

#### Act_OptP1030Del.st
```iecst
ACTION Act_OptP1030Del:

	IF tyP1030MagSet.tyMagSet.tyBtnDelete.bRtCompl = TRUE THEN
		IF usiDelMagRcpStep = 0 THEN
			tyP1030MagSet.tyMagSet.tyTableRecipe.uiMaskRtStat					:= FALSE;

			IF tyP1030MagSet.tyMagSet.tyTableRecipe.a_tyStringDataCol1[tyP1030Table.uiSelectedRow].sValue = p_tyMagRcpCurrRcp.sRcpNm THEN
				p_tyC0008MsgBox ACCESS ADR(tyP1030MagSet.tyMsgBoxDelCurrRcpAsk);

				IF tyP1030MagSet.tyMsgBoxDelCurrRcpAsk.tyBtnNo.bRtCompl = TRUE THEN
					tyP1030MagSet.tyMsgBoxDelCurrRcpAsk.tyBtnNo.bRtCompl 	:= FALSE;
					tyP1030MagSet.tyMsgBoxDelCurrRcpAsk.tyBtnNo.bValue 		:= FALSE;

					p_tyC0008MsgBox ACCESS ADR(tyP1030MagSet.tyMsgBoxHide);

					usiDelMagRcpStep	:= 99;
				END_IF
			ELSE
				p_tyC0008MsgBox ACCESS ADR(tyP1030MagSet.tyMsgBoxDelAsk);

				IF tyP1030MagSet.tyMsgBoxDelAsk.tyBtnYes.bRtCompl = TRUE THEN
					tyP1030MagSet.tyMsgBoxDelAsk.tyBtnYes.bRtCompl				:= FALSE;
					tyP1030MagSet.tyMsgBoxDelAsk.tyBtnYes.bValue				:= FALSE;

					p_tyC0008MsgBox ACCESS ADR(tyP1030MagSet.tyMsgBoxHide);

					usiDelMagRcpStep	:= 1;

				ELSIF tyP1030MagSet.tyMsgBoxDelAsk.tyBtnNo.bRtCompl = TRUE THEN
					tyP1030MagSet.tyMsgBoxDelAsk.tyBtnNo.bRtCompl			:= FALSE;
					tyP1030MagSet.tyMsgBoxDelAsk.tyBtnNo.bValue				:= FALSE;

					p_tyC0008MsgBox ACCESS ADR(tyP1030MagSet.tyMsgBoxHide);

					usiDelMagRcpStep	:= 99;

				END_IF
			END_IF

		ELSIF usiDelMagRcpStep = 1 THEN
			tyMagRcpInfoIn.sRcpNm			:= tyP1030MagSet.tyMagSet.tyTableRecipe.a_tyStringDataCol1[tyP1030Table.uiSelectedRow].sValue;

			eMagRcpAct					:= MagRcpActDel;

			IF p_eMagRcpStat = MagRcpActDel AND p_eMagRcpStatus = Done THEN
				eMagRcpAct				:= MagRcpActIdle;

				IF p_bMagRcpNmEmpty = TRUE THEN
					usiDelMagRcpStep		:= 2;
				ELSIF p_bMagRcpNmNotExist = TRUE THEN
					usiDelMagRcpStep		:= 3;
				ELSE
					tyP1030MagSet.tyMagSet.tyBtnSort.bValue	:= FALSE;
					bRefreshMagRcpTable		:= TRUE;
					bRefreshMagRcpDetail	:= TRUE;
					usiDelMagRcpStep		:= 99;
				END_IF

			ELSIF p_eMagRcpStatus = Error THEN
				p_tyC0008MsgBox ACCESS ADR(tyP1030MagSet.tyMsgBoxDelErr);

				IF tyP1030MagSet.tyMsgBoxDelErr.tyBtnNo.bRtCompl = TRUE THEN
					tyP1030MagSet.tyMsgBoxDelErr.tyBtnNo.bRtCompl 				:= FALSE;
					tyP1030MagSet.tyMsgBoxDelErr.tyBtnNo.bValue 				:= FALSE;

					p_tyC0008MsgBox ACCESS ADR(tyP1030MagSet.tyMsgBoxHide);

					usiDelMagRcpStep		:= 99;
				END_IF
			END_IF

		ELSIF usiDelMagRcpStep = 2 THEN
			p_tyC0008MsgBox ACCESS ADR(tyP1030MagSet.tyMsgBoxDelNmEmpty);

			IF tyP1030MagSet.tyMsgBoxDelNmEmpty.tyBtnNo.bRtCompl = TRUE THEN
				tyP1030MagSet.tyMsgBoxDelNmEmpty.tyBtnNo.bRtCompl 				:= FALSE;
				tyP1030MagSet.tyMsgBoxDelNmEmpty.tyBtnNo.bValue 				:= FALSE;

				p_tyC0008MsgBox ACCESS ADR(tyP1030MagSet.tyMsgBoxHide);

				usiDelMagRcpStep		:= 99;
			END_IF

		ELSIF usiDelMagRcpStep = 3 THEN
			p_tyC0008MsgBox ACCESS ADR(tyP1030MagSet.tyMsgBoxDelNmNotExist);

			IF tyP1030MagSet.tyMsgBoxDelNmNotExist.tyBtnNo.bRtCompl = TRUE THEN
				tyP1030MagSet.tyMsgBoxDelNmNotExist.tyBtnNo.bRtCompl 	:= FALSE;
				tyP1030MagSet.tyMsgBoxDelNmNotExist.tyBtnNo.bValue 		:= FALSE;

				p_tyC0008MsgBox ACCESS ADR(tyP1030MagSet.tyMsgBoxHide);

				usiDelMagRcpStep	:= 99;
			END_IF

		ELSIF usiDelMagRcpStep = 99 THEN
			bRefreshMagRcpTable	:= FALSE;

			//Unmask
			tyP1030MagSet.tyMagSet.tyTableRecipe.uiMaskRtStat			:= TRUE;

			//Reset
			tyP1030MagSet.tyMagSet.tyBtnDelete.bRtCompl					:= FALSE;
			tyP1030MagSet.tyMagSet.tyBtnDelete.bValue					:= FALSE;

			usiDelMagRcpStep		:= 0;
		END_IF

	END_IF

END_ACTION
```

#### Act_OptP1030Table.st
```iecst
ACTION Act_OptP1030Table:

	//Call Table FB
	fbP1030Table.sVisuNm			:= tyP1030Table.sVisuNm;
	fbP1030Table.udiWorkAreaStartX	:= 386;
	fbP1030Table.udiWorkAreaEndX	:= 796;
	fbP1030Table.udiWorkAreaStartY	:= 85;
	fbP1030Table.udiWorkAreaEndY	:= 405;
	fbP1030Table.udiMinXDist		:= 20;
	fbP1030Table.udiMinYDist		:= 20;
	fbP1030Table.uiSlideScale		:= c_uiP1030TableSize;
	fbP1030Table.iTotalData			:= UDINT_TO_INT(c_udiMagRcpMax);
	fbP1030Table.iTotalRow			:= c_uiP1030TableSize;
	fbP1030Table.p_uiSliderStatus	:= ADR(tyP1030MagSet.tyMagSet.tyTableRecipe.tyUISlider.uiRtStat);
	fbP1030Table.pa_tyUIHotspot		:= ADR(tyP1030MagSet.tyMagSet.tyTableRecipe.a_tyHotspot);
	fbP1030Table.p_uiTablePos		:= ADR(tyP1030Table.uiTablePos);
	fbP1030Table.p_iSliderPos		:= ADR(tyP1030MagSet.tyMagSet.tyTableRecipe.tyUISlider.iValue);
	fbP1030Table.p_uiSelectedRow	:= ADR(tyP1030Table.uiSelectedRow);
	fbP1030Table.p_bTableActive		:= ADR(tyP1030Table.bTableActive);
	fbP1030Table.p_bSliderActive	:= ADR(tyP1030Table.bSliderActive);
	fbP1030Table;

	//Table Content
	IF tyP1030Table.bTableActive = TRUE OR tyP1030Table.bSliderActive = TRUE OR bRefreshMagRcpTable = TRUE OR bUpdateP1030Table THEN
		FOR i := 1 TO c_uiP1030TableSize DO
			IF tyP1030MagSet.tyMagSet.tyBtnSort.bValue THEN
				tyP1030MagSet.tyMagSet.tyTableRecipe.a_tyStringDataCol0[i].sValue	    := UINT_TO_STRING(tyP1030Table.uiTablePos + i - 1);
				tyP1030MagSet.tyMagSet.tyTableRecipe.a_tyStringDataCol1[i].sValue		:= p_tyMagRcpSortedList[tyP1030Table.uiTablePos + i - 1].sRcpNm;
				tyP1030MagSet.tyMagSet.tyTableRecipe.a_tyStringDataCol2[i].sValue		:= p_tyMagRcpSortedList[tyP1030Table.uiTablePos + i - 1].sDisplayInfo;
			ELSE
				tyP1030MagSet.tyMagSet.tyTableRecipe.a_tyStringDataCol0[i].sValue	    := UINT_TO_STRING(tyP1030Table.uiTablePos + i - 1);
				tyP1030MagSet.tyMagSet.tyTableRecipe.a_tyStringDataCol1[i].sValue		:= p_tyMagRcpCurrList[tyP1030Table.uiTablePos + i - 1].sRcpNm;
				tyP1030MagSet.tyMagSet.tyTableRecipe.a_tyStringDataCol2[i].sValue		:= p_tyMagRcpCurrList[tyP1030Table.uiTablePos + i - 1].sDisplayInfo;
			END_IF
		END_FOR

		IF bUpdateP1030Table THEN
			bUpdateP1030Table := FALSE;
		END_IF
	END_IF

	//Selected Row
	IF tyP1030Table.uiSelectedRow <> tyP1030Table.uiSelectedRowOld THEN
		FOR i := 1 TO c_uiP1030TableSize DO
			IF tyP1030Table.uiSelectedRow = i THEN
				tyP1030MagSet.tyMagSet.tyTableRecipe.a_tyStringDataCol1[i].usiColor	:= 1;
				tyP1030MagSet.tyMagSet.tyTableRecipe.a_tyStringDataCol2[i].usiColor	:= 1;
			ELSE
				tyP1030MagSet.tyMagSet.tyTableRecipe.a_tyStringDataCol1[i].usiColor	:= 0;
				tyP1030MagSet.tyMagSet.tyTableRecipe.a_tyStringDataCol2[i].usiColor	:= 0;
			END_IF
		END_FOR

		tyP1030Table.uiSelectedRowOld	:= tyP1030Table.uiSelectedRow;
	END_IF

END_ACTION
```

#### Act_OptP1030Keypad.st
```iecst
ACTION Act_OptP1030Keypad:

	IF fUIOutRtStatTPIsOpen(ADR(tyP1030MagSet.tyMagSet.tyStringRecipeNm.uiRtStat)) THEN
		tyProperty.tyKeypad.tyStringTitle.sKeypadTitle	:= tyP1030MagSet.tyMagSet.tyStringRecipeNm.sKeypadTitle;

	ELSIF fUIOutRtStatTPIsOpen(ADR(tyP1030MagSet.tyMagSet.tyNumSltToSltDist.uiRtStat)) THEN
		tyProperty.tyKeypad.tyStringTitle.sKeypadTitle	:= tyP1030MagSet.tyMagSet.tyNumSltToSltDist.sKeypadTitle;

	ELSIF fUIOutRtStatTPIsOpen(ADR(tyP1030MagSet.tyMagSet.tyNumMaxSlt.uiRtStat)) THEN
		tyProperty.tyKeypad.tyStringTitle.sKeypadTitle	:= tyP1030MagSet.tyMagSet.tyNumMaxSlt.sKeypadTitle;

	ELSIF fUIOutRtStatTPIsOpen(ADR(tyP1030MagSet.tyMagSet.tyNumLifterMag1Slt1Pos.uiRtStat)) THEN
		tyProperty.tyKeypad.tyStringTitle.sKeypadTitle	:= tyP1030MagSet.tyMagSet.tyNumLifterMag1Slt1Pos.sKeypadTitle;

	ELSIF fUIOutRtStatTPIsOpen(ADR(tyP1030MagSet.tyMagSet.tyNumLifterMag2Slt1Pos.uiRtStat)) THEN
		tyProperty.tyKeypad.tyStringTitle.sKeypadTitle	:= tyP1030MagSet.tyMagSet.tyNumLifterMag2Slt1Pos.sKeypadTitle;

	ELSIF fUIOutRtStatTPIsOpen(ADR(tyP1030MagSet.tyMagSet.tyNumLifterMag3Slt1Pos.uiRtStat)) THEN
		tyProperty.tyKeypad.tyStringTitle.sKeypadTitle	:= tyP1030MagSet.tyMagSet.tyNumLifterMag3Slt1Pos.sKeypadTitle;

	ELSIF fUIOutRtStatTPIsOpen(ADR(tyP1030MagSet.tyMagSet.tyNumTravPosMag1.uiRtStat)) THEN
		tyProperty.tyKeypad.tyStringTitle.sKeypadTitle	:= tyP1030MagSet.tyMagSet.tyNumTravPosMag1.sKeypadTitle;

	ELSIF fUIOutRtStatTPIsOpen(ADR(tyP1030MagSet.tyMagSet.tyNumTravPosMag2.uiRtStat)) THEN
		tyProperty.tyKeypad.tyStringTitle.sKeypadTitle	:= tyP1030MagSet.tyMagSet.tyNumTravPosMag2.sKeypadTitle;

	ELSIF fUIOutRtStatTPIsOpen(ADR(tyP1030MagSet.tyMagSet.tyNumTravPosMag3.uiRtStat)) THEN
		tyProperty.tyKeypad.tyStringTitle.sKeypadTitle	:= tyP1030MagSet.tyMagSet.tyNumTravPosMag3.sKeypadTitle;

	ELSIF fUIOutRtStatTPIsOpen(ADR(tyP1030MagSet.tyMagSet.tyNumMagMaxBrdWidth.uiRtStat)) THEN
		tyProperty.tyKeypad.tyStringTitle.sKeypadTitle  := tyP1030MagSet.tyMagSet.tyNumMagMaxBrdWidth.sKeypadTitle;
	ELSE
		tyProperty.tyKeypad.tyStringTitle.sKeypadTitle	:= '';

	END_IF

END_ACTION
```

#### Act_OptP1030Teach.st
```iecst
ACTION Act_OptP1030Teach:

	IF tyP1030MagSet.tyMagSet.tyBtnLifterMag1Slt1Pos.bRtCompl = TRUE THEN
		tyP1030MagSet.tyMagSet.tyBtnLifterMag1Slt1Pos.bRtCompl	:= FALSE;
		tyP1030MagSet.tyMagSet.tyBtnLifterMag1Slt1Pos.bValue	:= FALSE;

		bTeachLifterMag1Slt1Pos	:= TRUE;
		eChgPage				:= UIP1031MagSetTeach;

	ELSIF tyP1030MagSet.tyMagSet.tyBtnLifterMag2Slt1Pos.bRtCompl = TRUE THEN
		tyP1030MagSet.tyMagSet.tyBtnLifterMag2Slt1Pos.bRtCompl	:= FALSE;
		tyP1030MagSet.tyMagSet.tyBtnLifterMag2Slt1Pos.bValue	:= FALSE;

		bTeachLifterMag2Slt1Pos	:= TRUE;
		eChgPage				:= UIP1031MagSetTeach;

	ELSIF tyP1030MagSet.tyMagSet.tyBtnLifterMag3Slt1Pos.bRtCompl = TRUE THEN
		tyP1030MagSet.tyMagSet.tyBtnLifterMag3Slt1Pos.bRtCompl	:= FALSE;
		tyP1030MagSet.tyMagSet.tyBtnLifterMag3Slt1Pos.bValue	:= FALSE;

		bTeachLifterMag3Slt1Pos	:= TRUE;
		eChgPage				:= UIP1031MagSetTeach;

	ELSIF tyP1030MagSet.tyMagSet.tyBtnTravPosMag1.bRtCompl = TRUE THEN
		tyP1030MagSet.tyMagSet.tyBtnTravPosMag1.bRtCompl	:= FALSE;
		tyP1030MagSet.tyMagSet.tyBtnTravPosMag1.bValue		:= FALSE;

		bTeachTravPosMag1	:= TRUE;
		eChgPage			:= UIP1031MagSetTeach;

	ELSIF tyP1030MagSet.tyMagSet.tyBtnTravPosMag2.bRtCompl = TRUE THEN
		tyP1030MagSet.tyMagSet.tyBtnTravPosMag2.bRtCompl	:= FALSE;
		tyP1030MagSet.tyMagSet.tyBtnTravPosMag2.bValue		:= FALSE;

		bTeachTravPosMag2	:= TRUE;
		eChgPage			:= UIP1031MagSetTeach;

	ELSIF tyP1030MagSet.tyMagSet.tyBtnTravPosMag3.bRtCompl = TRUE THEN
		tyP1030MagSet.tyMagSet.tyBtnTravPosMag3.bRtCompl	:= FALSE;
		tyP1030MagSet.tyMagSet.tyBtnTravPosMag3.bValue		:= FALSE;

		bTeachTravPosMag3	:= TRUE;
		eChgPage			:= UIP1031MagSetTeach;

	END_IF

END_ACTION
```

#### Act_OptP1030Sort.st
```iecst
ACTION Act_OptP1030Sort:

	IF tyP1030MagSet.tyMagSet.tyBtnSort.bValue THEN
		tyP1030MagSet.tyMagSet.tyBtnSort.usiTxtIdx 	:= 1;
	ELSE
		tyP1030MagSet.tyMagSet.tyBtnSort.usiTxtIdx 	:= 0;
	END_IF

	IF tyP1030MagSet.tyMagSet.tyBtnSort.bRtCompl THEN
		bUpdateP1030LoadData := TRUE;
	END_IF

	IF tyP1030MagSet.tyMagSet.tyBtnSort.bRtCompl THEN

		IF tyP1030MagSet.tyMagSet.tyBtnSort.bValue THEN

			tyP1030MagSet.tyMagSet.tyTableRecipe.uiMaskRtStat.0	:= FALSE;

			eMagRcpAct	:= MagRcpActSort;

			IF p_eMagRcpStat = MagRcpActSort AND p_eMagRcpStatus = Done THEN
				eMagRcpAct		:= MagRcpActIdle;

				FOR i := 1 TO c_uiP1030TableSize DO
					tyP1030MagSet.tyMagSet.tyTableRecipe.a_tyStringDataCol0[i].sValue	:= UINT_TO_STRING(tyP1030Table.uiTablePos + i - 1);
					tyP1030MagSet.tyMagSet.tyTableRecipe.a_tyStringDataCol1[i].sValue	:= p_tyMagRcpSortedList[tyP1030Table.uiTablePos + i - 1].sRcpNm;
					tyP1030MagSet.tyMagSet.tyTableRecipe.a_tyStringDataCol2[i].sValue	:= p_tyMagRcpSortedList[tyP1030Table.uiTablePos + i - 1].sDisplayInfo;
				END_FOR

				//Unmask
				tyP1030MagSet.tyMagSet.tyTableRecipe.uiMaskRtStat.0	:= TRUE;

				tyP1030MagSet.tyMagSet.tyBtnSort.bRtCompl := FALSE;

			ELSIF p_eMagRcpStatus = Error THEN
				FOR i := 1 TO c_uiP1030TableSize DO
					tyP1030MagSet.tyMagSet.tyTableRecipe.a_tyStringDataCol0[i].sValue		:= UINT_TO_STRING(tyP1030Table.uiTablePos + i - 1);
					tyP1030MagSet.tyMagSet.tyTableRecipe.a_tyStringDataCol1[i].sValue		:= '';
					tyP1030MagSet.tyMagSet.tyTableRecipe.a_tyStringDataCol2[i].sValue		:= '';
				END_FOR

				p_tyC0008MsgBox ACCESS ADR (tyP1030MagSet.tyMsgBoxListErr);

				IF tyP1030MagSet.tyMsgBoxListErr.tyBtnNo.bRtCompl = TRUE THEN
					tyP1030MagSet.tyMsgBoxListErr.tyBtnNo.bRtCompl 		:= TRUE;
					tyP1030MagSet.tyMsgBoxListErr.tyBtnNo.bValue			:= TRUE;

					p_tyC0008MsgBox ACCESS ADR (tyP1030MagSet.tyMsgBoxHide);

					//Unmask
					tyP1030MagSet.tyMagSet.tyTableRecipe.uiMaskRtStat.0	:= TRUE;

					//Reset
					tyP1030MagSet.tyMagSet.tyBtnSort.bRtCompl := FALSE;
				END_IF
			END_IF

		ELSE

			bUpdateP1030Table	:= TRUE;

			tyP1030MagSet.tyMagSet.tyBtnSort.bRtCompl := FALSE;

		END_IF

	END_IF

END_ACTION
```

#### Act_EntP1031Disp.st
```iecst
ACTION Act_EntP1031Disp:

	//Access Address
	p_tyC0002FullMask ACCESS ADR(tyP1031MagSetTeach.tyFullMaskHide);

	p_tyC0004Navi ACCESS ADR(tyP1031MagSetTeach.tyNaviBack);

	p_tyC0005Main ACCESS ADR(tyCommon.tyMain);

	p_tyC0007Notif ACCESS ADR(tyCommon.tyNotif);

	p_tyC0008MsgBox ACCESS ADR(tyP1031MagSetTeach.tyMsgBoxHide);

	p_tyC0009Info ACCESS ADR(tyCommon.tyInfo);

	p_tyP1031InOutletShutterFB ACCESS ADR(tyP1031MagSetTeach.tyInOutletShutterFB);

	IF bTeachLifterMag1Slt1Pos = TRUE THEN
		tyP1031MagSetTeach.tyTeachLifterMag1Slt1Pos.tyNumNewSlt.diValue := 1;
		tyP1031MagSetTeach.tyTeachLifterMag1Slt1Pos.tyNumNewSlt.diValueMin := 1;
		tyP1031MagSetTeach.tyTeachLifterMag1Slt1Pos.tyNumNewSlt.diValueMax := tyP1030MagSet.tyMagSet.tyNumMaxSlt.diValue;

		p_tyP1031MagSetTeach ACCESS ADR(tyP1031MagSetTeach.tyTeachLifterMag1Slt1Pos);
		p_tyC0001MotionStd ACCESS ADR(tyP1031MagSetTeach.tyMotionStdLifter);

	ELSIF bTeachLifterMag2Slt1Pos = TRUE THEN
		tyP1031MagSetTeach.tyTeachLifterMag2Slt1Pos.tyNumNewSlt.diValue := 1;
		tyP1031MagSetTeach.tyTeachLifterMag2Slt1Pos.tyNumNewSlt.diValueMin := 1;
		tyP1031MagSetTeach.tyTeachLifterMag2Slt1Pos.tyNumNewSlt.diValueMax := tyP1030MagSet.tyMagSet.tyNumMaxSlt.diValue;

		p_tyP1031MagSetTeach ACCESS ADR(tyP1031MagSetTeach.tyTeachLifterMag2Slt1Pos);
		p_tyC0001MotionStd ACCESS ADR(tyP1031MagSetTeach.tyMotionStdLifter);

	ELSIF bTeachLifterMag3Slt1Pos = TRUE THEN
		tyP1031MagSetTeach.tyTeachLifterMag3Slt1Pos.tyNumNewSlt.diValue := 1;
		tyP1031MagSetTeach.tyTeachLifterMag3Slt1Pos.tyNumNewSlt.diValueMin := 1;
		tyP1031MagSetTeach.tyTeachLifterMag3Slt1Pos.tyNumNewSlt.diValueMax := tyP1030MagSet.tyMagSet.tyNumMaxSlt.diValue;

		p_tyP1031MagSetTeach ACCESS ADR(tyP1031MagSetTeach.tyTeachLifterMag3Slt1Pos);
		p_tyC0001MotionStd ACCESS ADR(tyP1031MagSetTeach.tyMotionStdLifter);

	ELSIF bTeachTravPosMag1 = TRUE THEN
		tyP1031MagSetTeach.tyTeachTravPosMag1.tyNumNewSlt.uiRtStat.0 := TRUE;

		p_tyP1031MagSetTeach ACCESS ADR(tyP1031MagSetTeach.tyTeachTravPosMag1);
		p_tyC0001MotionStd ACCESS ADR(tyP1031MagSetTeach.tyMotionStdTrav);

	ELSIF bTeachTravPosMag2 = TRUE THEN
		tyP1031MagSetTeach.tyTeachTravPosMag2.tyNumNewSlt.uiRtStat.0 := TRUE;

		p_tyP1031MagSetTeach ACCESS ADR(tyP1031MagSetTeach.tyTeachTravPosMag2);
		p_tyC0001MotionStd ACCESS ADR(tyP1031MagSetTeach.tyMotionStdTrav);

	ELSIF bTeachTravPosMag3 = TRUE THEN
		tyP1031MagSetTeach.tyTeachTravPosMag3.tyNumNewSlt.uiRtStat.0 := TRUE;

		p_tyP1031MagSetTeach ACCESS ADR(tyP1031MagSetTeach.tyTeachTravPosMag3);
		p_tyC0001MotionStd ACCESS ADR(tyP1031MagSetTeach.tyMotionStdTrav);

	END_IF

	//Display
	//Traverser
	tyP1031MagSetTeach.tyMotionStdTrav.tyBtnPwr.bValue	:= p_bTravPwrOn;

	//Lifter
	tyP1031MagSetTeach.tyMotionStdLifter.tyBtnPwr.bValue	:= p_bLifterBtmPwrOn;

END_ACTION
```

#### Act_ExitP1031.st
```iecst
ACTION Act_ExitP1031:

	usiChgPage	:= 1;

	//Manual Deactivated
	bManualMod	:= FALSE;

	//Reset UI
	bJogSlow				:= FALSE;
	bJogFast				:= FALSE;
	fbJogSlowToFastDlyTm.IN	:= FALSE;

	fbLmtRstTm(IN := FALSE);
	//bypass curtain sensor
	bBypCurtainSen := FALSE;
	bBypCurtainPBLED := FALSE;
	tyP1031MagSetTeach.tyTeachTravPosMag1.tyBtn4.bValue				:= FALSE;
	tyP1031MagSetTeach.tyTeachTravPosMag2.tyBtn4.bValue				:= FALSE;
	tyP1031MagSetTeach.tyTeachTravPosMag3.tyBtn4.bValue				:= FALSE;
	tyP1031MagSetTeach.tyTeachLifterMag1Slt1Pos.tyBtn4.bValue				:= FALSE;
	tyP1031MagSetTeach.tyTeachLifterMag2Slt1Pos.tyBtn4.bValue				:= FALSE;
	tyP1031MagSetTeach.tyTeachLifterMag3Slt1Pos.tyBtn4.bValue				:= FALSE;

	//Traverser
	tyP1031MagSetTeach.tyMotionStdTrav.tyBtnPwr.bRtCompl			:= FALSE;
	tyP1031MagSetTeach.tyMotionStdTrav.tyBtnStop.bRtCompl			:= FALSE;
	tyP1031MagSetTeach.tyMotionStdTrav.tyBtnOrigin.bRtCompl			:= FALSE;
	tyP1031MagSetTeach.tyMotionStdTrav.tyBtnRst.bRtCompl			:= FALSE;
	tyP1031MagSetTeach.tyMotionStdTrav.tyBtnMovAbs.bRtCompl			:= FALSE;
	tyP1031MagSetTeach.tyMotionStdTrav.tyBtnMovRel.bRtCompl			:= FALSE;
	tyP1031MagSetTeach.tyMotionStdTrav.tyBtnJogFront.bRtCompl		:= FALSE;
	tyP1031MagSetTeach.tyMotionStdTrav.tyBtnJogRear.bRtCompl		:= FALSE;

	tyP1031MagSetTeach.tyTeachTravPosMag1.tyBtn2.bRtCompl			:= FALSE;
	tyP1031MagSetTeach.tyTeachTravPosMag2.tyBtn2.bRtCompl			:= FALSE;
	tyP1031MagSetTeach.tyTeachTravPosMag3.tyBtn2.bRtCompl			:= FALSE;

	tyP1031MagSetTeach.tyMotionStdTrav.tyBtnPwr.bValue				:= FALSE;
	tyP1031MagSetTeach.tyMotionStdTrav.tyBtnStop.bValue				:= TRUE;
	tyP1031MagSetTeach.tyMotionStdTrav.tyBtnOrigin.bValue			:= FALSE;
	tyP1031MagSetTeach.tyMotionStdTrav.tyBtnRst.bValue				:= FALSE;
	tyP1031MagSetTeach.tyMotionStdTrav.tyBtnMovAbs.bValue			:= FALSE;
	tyP1031MagSetTeach.tyMotionStdTrav.tyBtnMovRel.bValue			:= FALSE;
	tyP1031MagSetTeach.tyMotionStdTrav.tyBtnJogFront.bValue			:= FALSE;
	tyP1031MagSetTeach.tyMotionStdTrav.tyBtnJogRear.bValue			:= FALSE;

	tyP1031MagSetTeach.tyTeachTravPosMag1.tyBtn2.bValue				:= FALSE;
	tyP1031MagSetTeach.tyTeachTravPosMag2.tyBtn2.bValue				:= FALSE;
	tyP1031MagSetTeach.tyTeachTravPosMag3.tyBtn2.bValue				:= FALSE;

	tyP1031MagSetTeach.tyMotionStdTrav.tyBtnPwr.bRtLk				:= FALSE;
	tyP1031MagSetTeach.tyMotionStdTrav.tyBtnStop.bRtLk				:= TRUE;
	tyP1031MagSetTeach.tyMotionStdTrav.tyBtnOrigin.bRtLk			:= FALSE;
	tyP1031MagSetTeach.tyMotionStdTrav.tyBtnRst.bRtLk				:= FALSE;
	tyP1031MagSetTeach.tyMotionStdTrav.tyBtnMovAbs.bRtLk			:= FALSE;
	tyP1031MagSetTeach.tyMotionStdTrav.tyBtnMovRel.bRtLk			:= FALSE;
	tyP1031MagSetTeach.tyMotionStdTrav.tyBtnJogFront.bRtLk			:= FALSE;
	tyP1031MagSetTeach.tyMotionStdTrav.tyBtnJogRear.bRtLk			:= FALSE;

	tyP1031MagSetTeach.tyTeachTravPosMag1.tyBtn2.bRtLk				:= FALSE;
	tyP1031MagSetTeach.tyTeachTravPosMag2.tyBtn2.bRtLk				:= FALSE;
	tyP1031MagSetTeach.tyTeachTravPosMag3.tyBtn2.bRtLk				:= FALSE;

	tyP1031MagSetTeach.tyMotionStdTrav.tyBtnPwr.uiMaskRtStat		:= TRUE;
	tyP1031MagSetTeach.tyMotionStdTrav.tyBtnOrigin.uiMaskRtStat		:= FALSE;
	tyP1031MagSetTeach.tyMotionStdTrav.tyBtnRst.uiMaskRtStat		:= TRUE;
	tyP1031MagSetTeach.tyMotionStdTrav.tyBtnMovAbs.uiMaskRtStat		:= FALSE;
	tyP1031MagSetTeach.tyMotionStdTrav.tyBtnMovRel.uiMaskRtStat		:= FALSE;
	tyP1031MagSetTeach.tyMotionStdTrav.tyBtnJogFront.uiMaskRtStat	:= FALSE;
	tyP1031MagSetTeach.tyMotionStdTrav.tyBtnJogRear.uiMaskRtStat	:= FALSE;

	tyP1031MagSetTeach.tyTeachTravPosMag1.tyBtn2.uiMaskRtStat		:= FALSE;
	tyP1031MagSetTeach.tyTeachTravPosMag2.tyBtn2.uiMaskRtStat		:= FALSE;
	tyP1031MagSetTeach.tyTeachTravPosMag3.tyBtn2.uiMaskRtStat		:= FALSE;

	//Lifter
	tyP1031MagSetTeach.tyMotionStdLifter.tyBtnPwr.bRtCompl			:= FALSE;
	tyP1031MagSetTeach.tyMotionStdLifter.tyBtnStop.bRtCompl			:= FALSE;
	tyP1031MagSetTeach.tyMotionStdLifter.tyBtnOrigin.bRtCompl		:= FALSE;
	tyP1031MagSetTeach.tyMotionStdLifter.tyBtnRst.bRtCompl			:= FALSE;
	tyP1031MagSetTeach.tyMotionStdLifter.tyBtnMovAbs.bRtCompl		:= FALSE;
	tyP1031MagSetTeach.tyMotionStdLifter.tyBtnMovRel.bRtCompl		:= FALSE;
	tyP1031MagSetTeach.tyMotionStdLifter.tyBtnJogUp.bRtCompl		:= FALSE;
	tyP1031MagSetTeach.tyMotionStdLifter.tyBtnJogDown.bRtCompl		:= FALSE;

	tyP1031MagSetTeach.tyTeachLifterMag1Slt1Pos.tyBtn2.bRtCompl		:= FALSE;
	tyP1031MagSetTeach.tyTeachLifterMag2Slt1Pos.tyBtn2.bRtCompl		:= FALSE;
	tyP1031MagSetTeach.tyTeachLifterMag3Slt1Pos.tyBtn2.bRtCompl		:= FALSE;

	tyP1031MagSetTeach.tyMotionStdLifter.tyBtnPwr.bValue			:= FALSE;
	tyP1031MagSetTeach.tyMotionStdLifter.tyBtnStop.bValue			:= TRUE;
	tyP1031MagSetTeach.tyMotionStdLifter.tyBtnOrigin.bValue			:= FALSE;
	tyP1031MagSetTeach.tyMotionStdLifter.tyBtnRst.bValue			:= FALSE;
	tyP1031MagSetTeach.tyMotionStdLifter.tyBtnMovAbs.bValue			:= FALSE;
	tyP1031MagSetTeach.tyMotionStdLifter.tyBtnMovRel.bValue			:= FALSE;
	tyP1031MagSetTeach.tyMotionStdLifter.tyBtnJogUp.bValue			:= FALSE;
	tyP1031MagSetTeach.tyMotionStdLifter.tyBtnJogDown.bValue		:= FALSE;

	tyP1031MagSetTeach.tyTeachLifterMag1Slt1Pos.tyBtn2.bValue		:= FALSE;
	tyP1031MagSetTeach.tyTeachLifterMag2Slt1Pos.tyBtn2.bValue		:= FALSE;
	tyP1031MagSetTeach.tyTeachLifterMag3Slt1Pos.tyBtn2.bValue		:= FALSE;

	tyP1031MagSetTeach.tyMotionStdLifter.tyBtnPwr.bRtLk				:= FALSE;
	tyP1031MagSetTeach.tyMotionStdLifter.tyBtnStop.bRtLk			:= TRUE;
	tyP1031MagSetTeach.tyMotionStdLifter.tyBtnOrigin.bRtLk			:= FALSE;
	tyP1031MagSetTeach.tyMotionStdLifter.tyBtnRst.bRtLk				:= FALSE;
	tyP1031MagSetTeach.tyMotionStdLifter.tyBtnMovAbs.bRtLk			:= FALSE;
	tyP1031MagSetTeach.tyMotionStdLifter.tyBtnMovRel.bRtLk			:= FALSE;
	tyP1031MagSetTeach.tyMotionStdLifter.tyBtnJogUp.bRtLk			:= FALSE;
	tyP1031MagSetTeach.tyMotionStdLifter.tyBtnJogDown.bRtLk			:= FALSE;

	tyP1031MagSetTeach.tyTeachLifterMag1Slt1Pos.tyBtn2.bRtLk		:= FALSE;
	tyP1031MagSetTeach.tyTeachLifterMag2Slt1Pos.tyBtn2.bRtLk		:= FALSE;
	tyP1031MagSetTeach.tyTeachLifterMag3Slt1Pos.tyBtn2.bRtLk		:= FALSE;

	tyP1031MagSetTeach.tyMotionStdLifter.tyBtnPwr.uiMaskRtStat		:= TRUE;
	tyP1031MagSetTeach.tyMotionStdLifter.tyBtnOrigin.uiMaskRtStat	:= FALSE;
	tyP1031MagSetTeach.tyMotionStdLifter.tyBtnRst.uiMaskRtStat		:= TRUE;
	tyP1031MagSetTeach.tyMotionStdLifter.tyBtnMovAbs.uiMaskRtStat	:= FALSE;
	tyP1031MagSetTeach.tyMotionStdLifter.tyBtnMovRel.uiMaskRtStat	:= FALSE;
	tyP1031MagSetTeach.tyMotionStdLifter.tyBtnJogUp.uiMaskRtStat	:= FALSE;
	tyP1031MagSetTeach.tyMotionStdLifter.tyBtnJogDown.uiMaskRtStat	:= FALSE;

	tyP1031MagSetTeach.tyTeachLifterMag1Slt1Pos.tyBtn2.uiMaskRtStat	:= FALSE;
	tyP1031MagSetTeach.tyTeachLifterMag2Slt1Pos.tyBtn2.uiMaskRtStat	:= FALSE;
	tyP1031MagSetTeach.tyTeachLifterMag3Slt1Pos.tyBtn2.uiMaskRtStat	:= FALSE;

END_ACTION
```

#### Act_OptP1031Navi.st
```iecst
ACTION Act_OptP1031Navi:

	IF tyP1031MagSetTeach.tyNaviBack.tyBtnBack.bRtCompl = TRUE THEN
		tyP1031MagSetTeach.tyNaviBack.tyBtnBack.bRtCompl	:= FALSE;
		tyP1031MagSetTeach.tyNaviBack.tyBtnBack.bValue		:= FALSE;

		eChgPage	:= UIP1030MagSet;
	END_IF

END_ACTION
```

#### Act_OptP1031FullMask.st
```iecst
ACTION Act_OptP1031FullMask:

	IF eCurrPage = UIP1031MagSetTeach THEN

		IF p_tyDI.bEStopSig = FALSE THEN
			p_tyC0002FullMask ACCESS ADR(tyP1031MagSetTeach.tyFullMaskEStop);

		ELSIF p_tyDI.bCoverSWSig = FALSE THEN
			p_tyC0002FullMask ACCESS ADR(tyP1031MagSetTeach.tyFullMaskCWSig);

		ELSIF p_tyDI.bSafetyRlySig = FALSE THEN
			p_tyC0002FullMask ACCESS ADR(tyP1031MagSetTeach.tyFullMaskSafetyRly);

		ELSIF (bTeachLifterMag1Slt1Pos OR bTeachLifterMag2Slt1Pos OR bTeachLifterMag3Slt1Pos) AND (p_tyDI.bLifterSafetyLmtSW1 = FALSE OR p_tyDI.bLifterSafetyLmtSW2 = FALSE) THEN
			p_tyC0002FullMask ACCESS ADR(tyP1031MagSetTeach.tyFullMaskSafetyLmtSW);

		ELSIF (bTeachLifterMag1Slt1Pos OR bTeachLifterMag2Slt1Pos OR bTeachLifterMag3Slt1Pos) AND p_tyDI.bLifterTimingBeltSen = FALSE THEN
			p_tyC0002FullMask ACCESS ADR(tyP1031MagSetTeach.tyFullMaskTimingBelt);

		ELSE
			p_tyC0002FullMask ACCESS ADR(tyP1031MagSetTeach.tyFullMaskHide);

		END_IF

	END_IF

END_ACTION
```

#### Act_OptP1031Mnl.st
```iecst
ACTION Act_OptP1031Mnl:

	bManualMod	:= p_tyDI.bSafetyRlySig;

END_ACTION
```

#### Act_OptP1031TravTeach.st
```iecst
ACTION Act_OptP1031TravTeach:

	IF tyP1031MagSetTeach.tyTeachTravPosMag1.tyBtn1.bRtCompl = TRUE THEN

		p_tyC0008MsgBox ACCESS ADR(tyP1031MagSetTeach.tyMsgBoxUpdtTravPosMag1);

		IF tyP1031MagSetTeach.tyMsgBoxUpdtTravPosMag1.tyBtnNo.bRtCompl THEN
			tyP1031MagSetTeach.tyMsgBoxUpdtTravPosMag1.tyBtnNo.bRtCompl := FALSE;
			tyP1031MagSetTeach.tyMsgBoxUpdtTravPosMag1.tyBtnNo.bValue 	:= FALSE;

			p_tyC0008MsgBox ACCESS ADR(tyP1031MagSetTeach.tyMsgBoxHide);

			//Write Actual Position To Magazine Setting.
			tyP1030MagSet.tyMagSet.tyNumTravPosMag1.diValue 	:= p_diTravActualPos;
			tyP1030MagSet.tyMagSet.tyNumTravPosMag1.bRtCompl	:= TRUE;

			//Back To Magazine Settings
			eChgPage	:= UIP1030MagSet;

			fUIInRtStatHide(ADR(tyP1030MagSet.tyMagSet.tyBtnSave.uiMaskRtStat));

			tyP1031MagSetTeach.tyTeachTravPosMag1.tyBtn1.bRtCompl	:= FALSE;
			tyP1031MagSetTeach.tyTeachTravPosMag1.tyBtn1.bValue		:= FALSE;

		END_IF

	ELSIF tyP1031MagSetTeach.tyTeachTravPosMag2.tyBtn1.bRtCompl = TRUE THEN

		p_tyC0008MsgBox ACCESS ADR(tyP1031MagSetTeach.tyMsgBoxUpdtTravPosMag2);

		IF tyP1031MagSetTeach.tyMsgBoxUpdtTravPosMag2.tyBtnNo.bRtCompl THEN
			tyP1031MagSetTeach.tyMsgBoxUpdtTravPosMag2.tyBtnNo.bRtCompl := FALSE;
			tyP1031MagSetTeach.tyMsgBoxUpdtTravPosMag2.tyBtnNo.bValue 	:= FALSE;

			p_tyC0008MsgBox ACCESS ADR(tyP1031MagSetTeach.tyMsgBoxHide);

			//Write Actual Position To Magazine Setting.
			tyP1030MagSet.tyMagSet.tyNumTravPosMag2.diValue		:= p_diTravActualPos;
			tyP1030MagSet.tyMagSet.tyNumTravPosMag2.bRtCompl	:= TRUE;

			//Back To Magazine Settings
			eChgPage	:= UIP1030MagSet;

			fUIInRtStatHide(ADR(tyP1030MagSet.tyMagSet.tyBtnSave.uiMaskRtStat));

			tyP1031MagSetTeach.tyTeachTravPosMag2.tyBtn1.bRtCompl	:= FALSE;
			tyP1031MagSetTeach.tyTeachTravPosMag2.tyBtn1.bValue		:= FALSE;

		END_IF

	ELSIF tyP1031MagSetTeach.tyTeachTravPosMag3.tyBtn1.bRtCompl = TRUE THEN

		p_tyC0008MsgBox ACCESS ADR(tyP1031MagSetTeach.tyMsgBoxUpdtTravPosMag3);

		IF tyP1031MagSetTeach.tyMsgBoxUpdtTravPosMag3.tyBtnNo.bRtCompl THEN
			tyP1031MagSetTeach.tyMsgBoxUpdtTravPosMag3.tyBtnNo.bRtCompl := FALSE;
			tyP1031MagSetTeach.tyMsgBoxUpdtTravPosMag3.tyBtnNo.bValue 	:= FALSE;

			p_tyC0008MsgBox ACCESS ADR(tyP1031MagSetTeach.tyMsgBoxHide);

			//Write Actual Position To Magazine Setting.
			tyP1030MagSet.tyMagSet.tyNumTravPosMag3.diValue 	:= p_diTravActualPos;
			tyP1030MagSet.tyMagSet.tyNumTravPosMag3.bRtCompl	:= TRUE;

			//Back To Magazine Settings
			eChgPage	:= UIP1030MagSet;

			fUIInRtStatHide(ADR(tyP1030MagSet.tyMagSet.tyBtnSave.uiMaskRtStat));

			tyP1031MagSetTeach.tyTeachTravPosMag3.tyBtn1.bRtCompl	:= FALSE;
			tyP1031MagSetTeach.tyTeachTravPosMag3.tyBtn1.bValue		:= FALSE;

		END_IF

	END_IF

END_ACTION
```

#### Act_OptP1031TravFBCtrl.st
```iecst
ACTION Act_OptP1031TravFBCtrl:

	fbJogSlowToFastDlyTm.PT			:= T#2s;
	fbJogSlowToFastDlyTm;
	fbLmtRstTm;

//	IF EDGEPOS((p_udiTravAxisErrID = 21570 OR p_udiTravAxisErrID = 21571)
	IF EDGEPOS((p_bTravFwdLmtSen OR p_bTravRevLmtSen OR p_udiTravAxisErrID = 21570 OR p_udiTravAxisErrID = 21571)
		AND tyP1031MagSetTeach.tyMotionStdTrav.tyBtnJogRear.bValue = FALSE
		AND tyP1031MagSetTeach.tyMotionStdTrav.tyBtnJogFront.bValue = FALSE) THEN
		fbLmtRstTm.IN				:= TRUE;
	END_IF

	IF fbLmtRstTm.Q = TRUE THEN
		tyP1031MagSetTeach.tyMotionStdTrav.tyBtnRst.bRtCompl		:= TRUE;
	END_IF

	IF (tyP1031MagSetTeach.tyMotionStdTrav.tyBtnJogFront.bValue = FALSE AND tyP1031MagSetTeach.tyMotionStdTrav.tyBtnJogRear.bValue = FALSE) AND (p_bTravJogging = TRUE) THEN
		bJogStopTrav	:= TRUE;
	END_IF

	IF tyP1031MagSetTeach.tyMotionStdTrav.tyBtnStop.bRtCompl = TRUE THEN
		eTravAct		:= TravActStop;

		IF p_eTravStat = TravActStop AND p_eTravStatus = Done THEN
			eTravAct	:= TravActIdle;

			tyP1031MagSetTeach.tyMotionStdTrav.tyBtnStop.bRtCompl		:= FALSE;
			tyP1031MagSetTeach.tyMotionStdTrav.tyBtnJogRear.bRtCompl	:= FALSE;
			tyP1031MagSetTeach.tyMotionStdTrav.tyBtnJogFront.bRtCompl	:= FALSE;
			tyP1031MagSetTeach.tyMotionStdTrav.tyBtnOrigin.bRtCompl		:= FALSE;
			tyP1031MagSetTeach.tyMotionStdTrav.tyBtnMovAbs.bRtCompl		:= FALSE;
			tyP1031MagSetTeach.tyMotionStdTrav.tyBtnMovRel.bRtCompl		:= FALSE;

			tyP1031MagSetTeach.tyTeachTravPosMag1.tyBtn2.bRtCompl		:= FALSE;
			tyP1031MagSetTeach.tyTeachTravPosMag2.tyBtn2.bRtCompl		:= FALSE;
			tyP1031MagSetTeach.tyTeachTravPosMag3.tyBtn2.bRtCompl		:= FALSE;

			tyP1031MagSetTeach.tyMotionStdTrav.tyBtnStop.bValue			:= TRUE;
			tyP1031MagSetTeach.tyMotionStdTrav.tyBtnJogRear.bValue		:= FALSE;
			tyP1031MagSetTeach.tyMotionStdTrav.tyBtnJogFront.bValue		:= FALSE;
			tyP1031MagSetTeach.tyMotionStdTrav.tyBtnOrigin.bValue		:= FALSE;
			tyP1031MagSetTeach.tyMotionStdTrav.tyBtnMovAbs.bValue		:= FALSE;
			tyP1031MagSetTeach.tyMotionStdTrav.tyBtnMovRel.bValue		:= FALSE;

			tyP1031MagSetTeach.tyTeachTravPosMag1.tyBtn2.bValue			:= FALSE;
			tyP1031MagSetTeach.tyTeachTravPosMag2.tyBtn2.bValue			:= FALSE;
			tyP1031MagSetTeach.tyTeachTravPosMag3.tyBtn2.bValue			:= FALSE;

			tyP1031MagSetTeach.tyMotionStdTrav.tyBtnStop.bRtLk			:= TRUE;
			tyP1031MagSetTeach.tyMotionStdTrav.tyBtnJogRear.bRtLk		:= FALSE;
			tyP1031MagSetTeach.tyMotionStdTrav.tyBtnJogFront.bRtLk		:= FALSE;
			tyP1031MagSetTeach.tyMotionStdTrav.tyBtnOrigin.bRtLk		:= FALSE;
			tyP1031MagSetTeach.tyMotionStdTrav.tyBtnMovAbs.bRtLk		:= FALSE;
			tyP1031MagSetTeach.tyMotionStdTrav.tyBtnMovRel.bRtLk		:= FALSE;

			tyP1031MagSetTeach.tyTeachTravPosMag1.tyBtn2.bRtLk			:= FALSE;
			tyP1031MagSetTeach.tyTeachTravPosMag2.tyBtn2.bRtLk			:= FALSE;
			tyP1031MagSetTeach.tyTeachTravPosMag3.tyBtn2.bRtLk			:= FALSE;
		END_IF

	ELSIF (tyP1031MagSetTeach.tyMotionStdTrav.tyBtnJogRear.bRtCompl = TRUE) OR (tyP1031MagSetTeach.tyMotionStdTrav.tyBtnJogFront.bRtCompl = TRUE) OR (bJogStopTrav = TRUE) THEN
		bJogSlow					:= FALSE;
		bJogFast					:= FALSE;
		fbJogSlowToFastDlyTm.IN		:= FALSE;

		eTravAct		:= TravActJogStop;

		IF p_eTravStat = TravActJogStop AND p_eTravStatus = Done THEN
			eTravAct		:= TravActIdle;

			bJogStopTrav	:= FALSE;

			tyP1031MagSetTeach.tyMotionStdTrav.tyBtnStop.bRtCompl		:= FALSE;
			tyP1031MagSetTeach.tyMotionStdTrav.tyBtnJogRear.bRtCompl	:= FALSE;
			tyP1031MagSetTeach.tyMotionStdTrav.tyBtnJogFront.bRtCompl	:= FALSE;
			tyP1031MagSetTeach.tyMotionStdTrav.tyBtnOrigin.bRtCompl		:= FALSE;
			tyP1031MagSetTeach.tyMotionStdTrav.tyBtnMovAbs.bRtCompl		:= FALSE;
			tyP1031MagSetTeach.tyMotionStdTrav.tyBtnMovRel.bRtCompl		:= FALSE;

			tyP1031MagSetTeach.tyTeachTravPosMag1.tyBtn2.bRtCompl		:= FALSE;
			tyP1031MagSetTeach.tyTeachTravPosMag2.tyBtn2.bRtCompl		:= FALSE;
			tyP1031MagSetTeach.tyTeachTravPosMag3.tyBtn2.bRtCompl		:= FALSE;

			tyP1031MagSetTeach.tyMotionStdTrav.tyBtnStop.bValue			:= TRUE;
			tyP1031MagSetTeach.tyMotionStdTrav.tyBtnJogRear.bValue		:= FALSE;
			tyP1031MagSetTeach.tyMotionStdTrav.tyBtnJogFront.bValue		:= FALSE;
			tyP1031MagSetTeach.tyMotionStdTrav.tyBtnOrigin.bValue		:= FALSE;
			tyP1031MagSetTeach.tyMotionStdTrav.tyBtnMovAbs.bValue		:= FALSE;
			tyP1031MagSetTeach.tyMotionStdTrav.tyBtnMovRel.bValue		:= FALSE;

			tyP1031MagSetTeach.tyTeachTravPosMag1.tyBtn2.bValue			:= FALSE;
			tyP1031MagSetTeach.tyTeachTravPosMag2.tyBtn2.bValue			:= FALSE;
			tyP1031MagSetTeach.tyTeachTravPosMag3.tyBtn2.bValue			:= FALSE;

			tyP1031MagSetTeach.tyMotionStdTrav.tyBtnStop.bRtLk			:= TRUE;
			tyP1031MagSetTeach.tyMotionStdTrav.tyBtnJogRear.bRtLk		:= FALSE;
			tyP1031MagSetTeach.tyMotionStdTrav.tyBtnJogFront.bRtLk		:= FALSE;
			tyP1031MagSetTeach.tyMotionStdTrav.tyBtnOrigin.bRtLk		:= FALSE;
			tyP1031MagSetTeach.tyMotionStdTrav.tyBtnMovAbs.bRtLk		:= FALSE;
			tyP1031MagSetTeach.tyMotionStdTrav.tyBtnMovRel.bRtLk		:= FALSE;

			tyP1031MagSetTeach.tyTeachTravPosMag1.tyBtn2.bRtLk			:= FALSE;
			tyP1031MagSetTeach.tyTeachTravPosMag2.tyBtn2.bRtLk			:= FALSE;
			tyP1031MagSetTeach.tyTeachTravPosMag3.tyBtn2.bRtLk			:= FALSE;

		END_IF

	ELSIF tyP1031MagSetTeach.tyMotionStdTrav.tyBtnPwr.bRtCompl = TRUE THEN
		tyP1031MagSetTeach.tyMotionStdTrav.tyBtnPwr.bRtLk				:= TRUE;

		IF tyP1031MagSetTeach.tyMotionStdTrav.tyBtnPwr.bValue = TRUE THEN
			eTravAct		:= TravActPwrOn;

			IF p_eTravStat = TravActPwrOn AND p_eTravStatus = Done THEN
				eTravAct	:= TravActIdle;

				tyP1031MagSetTeach.tyMotionStdTrav.tyBtnPwr.bRtCompl	:= FALSE;
				tyP1031MagSetTeach.tyMotionStdTrav.tyBtnPwr.bRtLk		:= FALSE;
			END_IF
		ELSE
			eTravAct		:= TravActPwrOff;

			IF p_eTravStat = TravActPwrOff AND p_eTravStatus = Done THEN
				eTravAct	:= TravActIdle;

				tyP1031MagSetTeach.tyMotionStdTrav.tyBtnPwr.bRtCompl		:= FALSE;
				tyP1031MagSetTeach.tyMotionStdTrav.tyBtnPwr.bRtLk		:= FALSE;
			END_IF
		END_IF

	ELSIF tyP1031MagSetTeach.tyMotionStdTrav.tyBtnOrigin.bRtCompl = TRUE THEN
		tyP1031MagSetTeach.tyMotionStdTrav.tyBtnOrigin.bValue			:= TRUE;
		tyP1031MagSetTeach.tyMotionStdTrav.tyBtnStop.bValue				:= FALSE;

		tyP1031MagSetTeach.tyMotionStdTrav.tyBtnOrigin.bRtLk				:= TRUE;
		tyP1031MagSetTeach.tyMotionStdTrav.tyBtnStop.bRtLk				:= FALSE;

		eTravAct		:= TravActHoming;

		IF p_eTravStat = TravActHoming AND p_eTravStatus = Done THEN
			eTravAct	:= TravActIdle;

			tyP1031MagSetTeach.tyMotionStdTrav.tyBtnOrigin.bRtCompl		:= FALSE;
			tyP1031MagSetTeach.tyMotionStdTrav.tyBtnOrigin.bValue		:= FALSE;
			tyP1031MagSetTeach.tyMotionStdTrav.tyBtnStop.bValue			:= TRUE;

			tyP1031MagSetTeach.tyMotionStdTrav.tyBtnOrigin.bRtLk		:= FALSE;
			tyP1031MagSetTeach.tyMotionStdTrav.tyBtnStop.bRtLk			:= TRUE;
		END_IF

	ELSIF tyP1031MagSetTeach.tyMotionStdTrav.tyBtnRst.bRtCompl = TRUE THEN
		tyP1031MagSetTeach.tyMotionStdTrav.tyBtnRst.bValue				:= TRUE;
		tyP1031MagSetTeach.tyMotionStdTrav.tyBtnRst.bRtLk				:= TRUE;

		eTravAct		:= TravActRstAxisErr;

		IF p_eTravStat = TravActRstAxisErr AND p_eTravStatus = Done THEN
			eTravAct	:= TravActIdle;

			tyP1031MagSetTeach.tyMotionStdTrav.tyBtnRst.bRtCompl		:= FALSE;
			tyP1031MagSetTeach.tyMotionStdTrav.tyBtnRst.bValue			:= FALSE;
			tyP1031MagSetTeach.tyMotionStdTrav.tyBtnRst.bRtLk			:= FALSE;

			fbLmtRstTm.IN			:= FALSE;
		END_IF

	ELSIF tyP1031MagSetTeach.tyTeachTravPosMag1.tyBtn2.bRtCompl = TRUE THEN
		tyP1031MagSetTeach.tyTeachTravPosMag1.tyBtn2.bValue		:= TRUE;
		tyP1031MagSetTeach.tyMotionStdTrav.tyBtnStop.bValue		:= FALSE;

		tyP1031MagSetTeach.tyTeachTravPosMag1.tyBtn2.bRtLk		:= TRUE;
		tyP1031MagSetTeach.tyMotionStdTrav.tyBtnStop.bRtLk		:= FALSE;

		diMnlTravNomSpd		:= tyP1031MagSetTeach.tyMotionStdTrav.tyNumNomSpd.diValue;

		eTravAct		:= TravActGoDPos;

		IF p_eTravStat = TravActGoDPos AND p_eTravStatus = Done THEN
			eTravAct	:= TravActIdle;

			tyP1031MagSetTeach.tyTeachTravPosMag1.tyBtn2.bRtCompl		:= FALSE;
			tyP1031MagSetTeach.tyTeachTravPosMag1.tyBtn2.bValue			:= FALSE;
			tyP1031MagSetTeach.tyMotionStdTrav.tyBtnStop.bValue			:= TRUE;

			tyP1031MagSetTeach.tyTeachTravPosMag1.tyBtn2.bRtLk			:= FALSE;
			tyP1031MagSetTeach.tyMotionStdTrav.tyBtnStop.bRtLk			:= TRUE;
		END_IF

	ELSIF tyP1031MagSetTeach.tyTeachTravPosMag2.tyBtn2.bRtCompl = TRUE THEN
		tyP1031MagSetTeach.tyTeachTravPosMag2.tyBtn2.bValue		:= TRUE;
		tyP1031MagSetTeach.tyMotionStdTrav.tyBtnStop.bValue		:= FALSE;

		tyP1031MagSetTeach.tyTeachTravPosMag2.tyBtn2.bRtLk		:= TRUE;
		tyP1031MagSetTeach.tyMotionStdTrav.tyBtnStop.bRtLk		:= FALSE;

		diMnlTravNomSpd		:= tyP1031MagSetTeach.tyMotionStdTrav.tyNumNomSpd.diValue;

		eTravAct		:= TravActGoEPos;

		IF p_eTravStat = TravActGoEPos AND p_eTravStatus = Done THEN
			eTravAct	:= TravActIdle;

			tyP1031MagSetTeach.tyTeachTravPosMag2.tyBtn2.bRtCompl		:= FALSE;
			tyP1031MagSetTeach.tyTeachTravPosMag2.tyBtn2.bValue			:= FALSE;
			tyP1031MagSetTeach.tyMotionStdTrav.tyBtnStop.bValue			:= TRUE;

			tyP1031MagSetTeach.tyTeachTravPosMag2.tyBtn2.bRtLk			:= FALSE;
			tyP1031MagSetTeach.tyMotionStdTrav.tyBtnStop.bRtLk			:= TRUE;
		END_IF

	ELSIF tyP1031MagSetTeach.tyTeachTravPosMag3.tyBtn2.bRtCompl = TRUE THEN
		tyP1031MagSetTeach.tyTeachTravPosMag3.tyBtn2.bValue		:= TRUE;
		tyP1031MagSetTeach.tyMotionStdTrav.tyBtnStop.bValue		:= FALSE;

		tyP1031MagSetTeach.tyTeachTravPosMag3.tyBtn2.bRtLk		:= TRUE;
		tyP1031MagSetTeach.tyMotionStdTrav.tyBtnStop.bRtLk		:= FALSE;

		diMnlTravNomSpd		:= tyP1031MagSetTeach.tyMotionStdTrav.tyNumNomSpd.diValue;

		eTravAct		:= TravActGoFPos;

		IF p_eTravStat = TravActGoFPos AND p_eTravStatus = Done THEN
			eTravAct	:= TravActIdle;

			tyP1031MagSetTeach.tyTeachTravPosMag3.tyBtn2.bRtCompl		:= FALSE;
			tyP1031MagSetTeach.tyTeachTravPosMag3.tyBtn2.bValue			:= FALSE;
			tyP1031MagSetTeach.tyMotionStdTrav.tyBtnStop.bValue			:= TRUE;

			tyP1031MagSetTeach.tyTeachTravPosMag3.tyBtn2.bRtLk			:= FALSE;
			tyP1031MagSetTeach.tyMotionStdTrav.tyBtnStop.bRtLk			:= TRUE;
		END_IF

	ELSIF tyP1031MagSetTeach.tyMotionStdTrav.tyBtnMovAbs.bRtCompl = TRUE THEN
		tyP1031MagSetTeach.tyMotionStdTrav.tyBtnMovAbs.bValue			:= TRUE;
		tyP1031MagSetTeach.tyMotionStdTrav.tyBtnStop.bValue				:= FALSE;

		tyP1031MagSetTeach.tyMotionStdTrav.tyBtnMovAbs.bRtLk				:= TRUE;
		tyP1031MagSetTeach.tyMotionStdTrav.tyBtnStop.bRtLk				:= FALSE;

		diMnlTravTargetPos	:= tyP1031MagSetTeach.tyMotionStdTrav.tyNumTargetPos.diValue;
		diMnlTravNomSpd		:= tyP1031MagSetTeach.tyMotionStdTrav.tyNumNomSpd.diValue;

		eTravAct		:= TravActMovAbs;

		IF p_eTravStat = TravActMovAbs AND p_eTravStatus = Done THEN
			eTravAct	:= TravActIdle;

			tyP1031MagSetTeach.tyMotionStdTrav.tyBtnMovAbs.bRtCompl		:= FALSE;
			tyP1031MagSetTeach.tyMotionStdTrav.tyBtnMovAbs.bValue		:= FALSE;
			tyP1031MagSetTeach.tyMotionStdTrav.tyBtnStop.bValue			:= TRUE;

			tyP1031MagSetTeach.tyMotionStdTrav.tyBtnMovAbs.bRtLk			:= FALSE;
			tyP1031MagSetTeach.tyMotionStdTrav.tyBtnStop.bRtLk			:= TRUE;
		END_IF

	ELSIF tyP1031MagSetTeach.tyMotionStdTrav.tyBtnMovRel.bRtCompl = TRUE THEN
		tyP1031MagSetTeach.tyMotionStdTrav.tyBtnMovRel.bValue			:= TRUE;
		tyP1031MagSetTeach.tyMotionStdTrav.tyBtnStop.bValue				:= FALSE;

		tyP1031MagSetTeach.tyMotionStdTrav.tyBtnMovRel.bRtLk				:= TRUE;
		tyP1031MagSetTeach.tyMotionStdTrav.tyBtnStop.bRtLk				:= FALSE;

		diMnlTravStepSize	:= tyP1031MagSetTeach.tyMotionStdTrav.tyNumStepSize.diValue;
		diMnlTravNomSpd		:= tyP1031MagSetTeach.tyMotionStdTrav.tyNumNomSpd.diValue;

		eTravAct		:= TravActMovRel;

		IF p_eTravStat = TravActMovRel AND p_eTravStatus = Done THEN
			eTravAct	:= TravActIdle;

			tyP1031MagSetTeach.tyMotionStdTrav.tyBtnMovRel.bRtCompl		:= FALSE;
			tyP1031MagSetTeach.tyMotionStdTrav.tyBtnMovRel.bValue		:= FALSE;
			tyP1031MagSetTeach.tyMotionStdTrav.tyBtnStop.bValue			:= TRUE;

			tyP1031MagSetTeach.tyMotionStdTrav.tyBtnMovRel.bRtLk			:= FALSE;
			tyP1031MagSetTeach.tyMotionStdTrav.tyBtnStop.bRtLk			:= TRUE;
		END_IF

	ELSIF (tyP1031MagSetTeach.tyMotionStdTrav.tyBtnJogRear.bValue = TRUE) AND (fbJogSlowToFastDlyTm.Q = FALSE) AND (bJogSlow = FALSE) THEN
		tyP1031MagSetTeach.tyMotionStdTrav.tyBtnStop.bValue				:= FALSE;
		tyP1031MagSetTeach.tyMotionStdTrav.tyBtnStop.bRtLk				:= FALSE;

		fbJogSlowToFastDlyTm.IN		:= TRUE;

		diMnlTravJogSpd	:= tyP1031MagSetTeach.tyMotionStdTrav.tyNumSlwSpd.diValue;

		eTravAct		:= TravActJogRear;

		IF p_eTravStat = TravActJogRear AND p_eTravStatus = Done THEN
			eTravAct	:= TravActIdle;
			bJogSlow				:= TRUE;
		ELSIF p_eTravStatus = Error THEN
			fbJogSlowToFastDlyTm.IN	:= FALSE;
			bJogSlow				:= TRUE;
		END_IF

	ELSIF (tyP1031MagSetTeach.tyMotionStdTrav.tyBtnJogRear.bValue = TRUE) AND (fbJogSlowToFastDlyTm.Q = TRUE) AND (bJogFast = FALSE) THEN
		tyP1031MagSetTeach.tyMotionStdTrav.tyBtnStop.bValue					:= FALSE;
		tyP1031MagSetTeach.tyMotionStdTrav.tyBtnStop.bRtLk					:= FALSE;

		fbJogSlowToFastDlyTm.IN		:= TRUE;

		diMnlTravJogSpd	:= tyP1031MagSetTeach.tyMotionStdTrav.tyNumNomSpd.diValue;

		eTravAct		:= TravActJogRear;

		IF p_eTravStat = TravActJogRear AND p_eTravStatus = Done THEN
			eTravAct	:= TravActIdle;
			bJogFast				:= TRUE;
		ELSIF p_eTravStatus = Error THEN
			fbJogSlowToFastDlyTm.IN	:= FALSE;
			bJogFast				:= TRUE;
		END_IF

	ELSIF (tyP1031MagSetTeach.tyMotionStdTrav.tyBtnJogFront.bValue = TRUE) AND (fbJogSlowToFastDlyTm.Q = FALSE) AND (bJogSlow = FALSE) THEN
		tyP1031MagSetTeach.tyMotionStdTrav.tyBtnStop.bValue				:= FALSE;
		tyP1031MagSetTeach.tyMotionStdTrav.tyBtnStop.bRtLk				:= FALSE;

		fbJogSlowToFastDlyTm.IN		:= TRUE;

		diMnlTravJogSpd	:= tyP1031MagSetTeach.tyMotionStdTrav.tyNumSlwSpd.diValue;

		eTravAct		:= TravActJogFront;

		IF p_eTravStat = TravActJogFront AND p_eTravStatus = Done THEN
			eTravAct	:= TravActIdle;
			bJogSlow				:= TRUE;
		ELSIF p_eTravStatus = Error THEN
			fbJogSlowToFastDlyTm.IN	:= FALSE;
			bJogSlow				:= TRUE;
		END_IF

	ELSIF (tyP1031MagSetTeach.tyMotionStdTrav.tyBtnJogFront.bValue = TRUE) AND (fbJogSlowToFastDlyTm.Q = TRUE) AND (bJogFast = FALSE) THEN
		tyP1031MagSetTeach.tyMotionStdTrav.tyBtnStop.bValue				:= FALSE;
		tyP1031MagSetTeach.tyMotionStdTrav.tyBtnStop.bRtLk				:= FALSE;

		fbJogSlowToFastDlyTm.IN		:= TRUE;

		diMnlTravJogSpd	:= tyP1031MagSetTeach.tyMotionStdTrav.tyNumNomSpd.diValue;

		eTravAct		:= TravActJogFront;

		IF p_eTravStat = TravActJogFront AND p_eTravStatus = Done THEN
			eTravAct	:= TravActIdle;
			bJogFast	:= TRUE;
		ELSIF p_eTravStatus = Error THEN
			fbJogSlowToFastDlyTm.IN	:= FALSE;
			bJogFast				:= TRUE;
		END_IF
	END_IF

	IF tyP1031MagSetTeach.tyInOutletShutterFB.tyBtnOpen.bValue = TRUE THEN
		eInShutterAct	:= PneuActRet;
		eOutShutterAct	:= PneuActRet;
		eOutShutterAct2 := PneuActRet;
		eOutShutterAct3 := PneuActRet;

		IF (p_eInShutterStat = PneuActRet AND p_eInShutterStatus = Done)
			AND (p_eOutShutterStat = PneuActRet AND p_eOutShutterStatus = Done)
			AND (p_eOutShutterStat2 = PneuActRet AND p_eOutShutterStatus2 = Done)
			AND (p_eOutShutterStat3 = PneuActRet AND p_eOutShutterStatus3 = Done)
			THEN
			eInShutterAct	:= PneuActIdle;
			eOutShutterAct	:= PneuActIdle;
			eOutShutterAct2	:= PneuActIdle;
			eOutShutterAct3	:= PneuActIdle;
			tyP1031MagSetTeach.tyInOutletShutterFB.tyBtnOpen.bValue	:= FALSE;
		ELSIF p_eInShutterStatus = Error OR p_eOutShutterStatus = Error OR p_eOutShutterStatus2 = Error OR p_eOutShutterStatus3 = Error THEN
			tyP1031MagSetTeach.tyInOutletShutterFB.tyBtnOpen.bValue	:= FALSE;
		END_IF

	ELSIF tyP1031MagSetTeach.tyInOutletShutterFB.tyBtnClose.bValue = TRUE THEN
		eInShutterAct	:= PneuActExt;
		eOutShutterAct	:= PneuActExt;
		eOutShutterAct2	:= PneuActExt;
		eOutShutterAct3	:= PneuActExt;
		IF (p_eInShutterStat = PneuActExt AND p_eInShutterStatus = Done)
			AND (p_eOutShutterStat = PneuActExt AND p_eOutShutterStatus = Done)
			AND (p_eOutShutterStat2 = PneuActExt AND p_eOutShutterStatus2 = Done)
			AND (p_eOutShutterStat3 = PneuActExt AND p_eOutShutterStatus3 = Done)

			THEN
			eInShutterAct	:= PneuActIdle;
			eOutShutterAct	:= PneuActIdle;
			eOutShutterAct2	:= PneuActIdle;
			eOutShutterAct3	:= PneuActIdle;
			tyP1031MagSetTeach.tyInOutletShutterFB.tyBtnClose.bValue := FALSE;
		ELSIF p_eInShutterStatus = Error OR p_eOutShutterStatus = Error THEN
			tyP1031MagSetTeach.tyInOutletShutterFB.tyBtnClose.bValue := FALSE;
		END_IF
	END_IF

	IF p_eTravStat = TravActJogStop AND (p_eTravStatus = Done OR p_eTravStatus = Error) THEN
		eTravAct		:= TravActIdle;
	END_IF

	//bypass curtain sensor
	IF bTeachTravPosMag1 OR bTeachTravPosMag2 OR bTeachTravPosMag3 THEN
		bBypCurtainSen			:= tyP1031MagSetTeach.tyTeachTravPosMag1.tyBtn4.bValue OR tyP1031MagSetTeach.tyTeachTravPosMag2.tyBtn4.bValue OR tyP1031MagSetTeach.tyTeachTravPosMag3.tyBtn4.bValue;
		bBypCurtainPBLED		:= tyP1031MagSetTeach.tyTeachTravPosMag1.tyBtn4.bValue OR tyP1031MagSetTeach.tyTeachTravPosMag2.tyBtn4.bValue OR tyP1031MagSetTeach.tyTeachTravPosMag3.tyBtn4.bValue;
	END_IF

END_ACTION
```

#### Act_OptP1031TravFBStat.st
```iecst
ACTION Act_OptP1031TravFBStat:

	IF p_bTravAxisErr = TRUE THEN
		tyP1031MagSetTeach.tyMotionStdTrav.tyStringStat.sValue		:= p_sTravAxisErrTxt;
	ELSE
		tyP1031MagSetTeach.tyMotionStdTrav.tyStringStat.sValue		:= p_sTravStatTxt;
	END_IF

END_ACTION
```
